ABB RAPID module: MonProgramme.mod

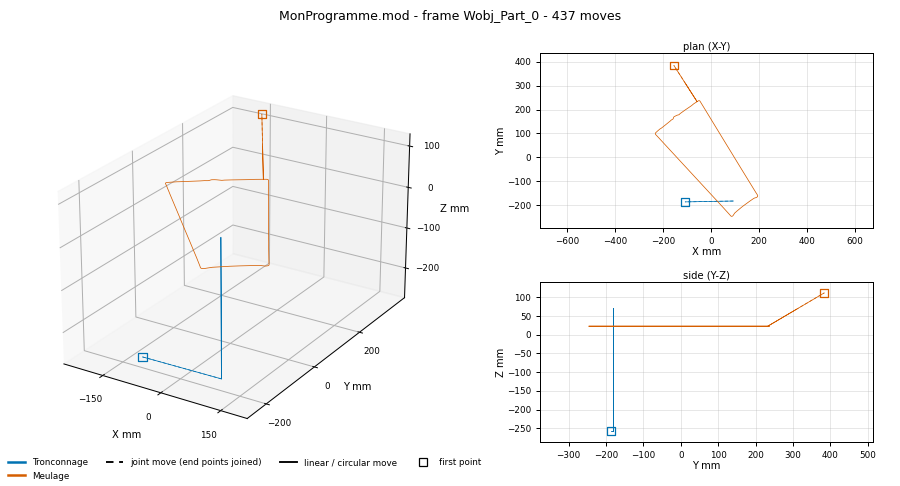
[picture p0: tool path of MonProgramme.mod in frame Wobj_Part_0, 437 of 442 moves have a stored position in this frame; points joined in program order, loops and branches not executed]
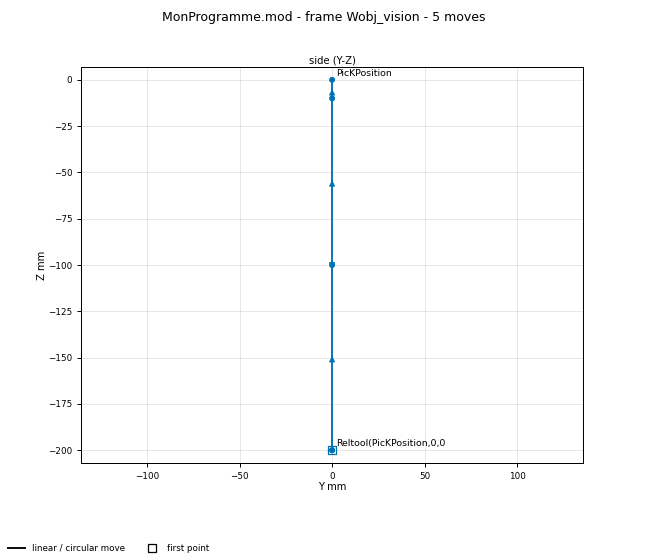
[picture p1: tool path of MonProgramme.mod in frame Wobj_vision, 5 of 442 moves have a stored position in this frame; points joined in program order, loops and branches not executed]
MODULE MonProgramme

    ! Nom         :MonProgramme
    ! Description :Pièce plate numero 1 famille 10
    ! Cree le     :30/03/2023 10:33:36

    CONST SPEEDDATA VitesseLente :=[10,500,0,0];
    CONST SPEEDDATA VitesseRapide :=[20,500,0,0];
    !
    !Point de prise
    PERS Robtarget PicKPosition := [[0,0,0],[0,0,0,0],[0,0,0,0],[9E9,9E9,9E9,9E9,9E9,9E9]];
    PERS Pose Ref := [[0,0,0],[1,0,0,0]];
    !
    !Declaration des points de meulage

    !Meulage_1 : Meulage du plan de joint
    CONST Robtarget Meulage_1_0 := [[-58.3575,232.789,23],[0.148181865705,-0.238974835253123,0.815584650429269,-0.505722098366382],[0,0,0,0],[8.999999E+09,8.999999E+09,8.999999E+09,8.999999E+09,8.999999E+09,8.999999E+09]];
    CONST Robtarget Meulage_1_1 := [[-61.8861,230.625,23],[0.148625433017615,-0.239693187884457,0.815376906988774,-0.505586941970947],[0,0,0,0],[8.999999E+09,8.999999E+09,8.999999E+09,8.999999E+09,8.999999E+09,8.999999E+09]];
    CONST Robtarget Meulage_1_2 := [[-62.4113,230.301,23],[0.149925832812002,-0.241798832684592,0.814763562882074,-0.505188980251654],[0,0,0,0],[8.999999E+09,8.999999E+09,8.999999E+09,8.999999E+09,8.999999E+09,8.999999E+09]];
    CONST Robtarget Meulage_1_3 := [[-62.698,230.118,23],[0.151989778330523,-0.245141375569821,0.81377802973829,-0.504549434230225],[0,0,0,0],[8.999999E+09,8.999999E+09,8.999999E+09,8.999999E+09,8.999999E+09,8.999999E+09]];
    CONST Robtarget Meulage_1_4 := [[-63.1019,229.854,23],[0.154659485743828,-0.249466287008623,0.812481437559476,-0.50370718551245],[0,0,0,0],[8.999999E+09,8.999999E+09,8.999999E+09,8.999999E+09,8.999999E+09,8.999999E+09]];
    CONST Robtarget Meulage_1_5 := [[-70.7437,224.925,23],[0.157674904224026,-0.254354542291001,0.810988113593647,-0.502733200618079],[0,0,0,0],[8.999999E+09,8.999999E+09,8.999999E+09,8.999999E+09,8.999999E+09,8.999999E+09]];
    CONST Robtarget Meulage_1_6 := [[-71.9304,224.189,23],[0.160716946471538,-0.259293185737598,0.80945258539058,-0.501720658286478],[0,0,0,0],[8.999999E+09,8.999999E+09,8.999999E+09,8.999999E+09,8.999999E+09,8.999999E+09]];
    CONST Robtarget Meulage_1_7 := [[-74.21,222.511,23],[0.163429453183647,-0.26370625584774,0.808060318676629,-0.500787725327893],[0,0,0,0],[8.999999E+09,8.999999E+09,8.999999E+09,8.999999E+09,8.999999E+09,8.999999E+09]];
    CONST Robtarget Meulage_1_8 := [[-74.4047,222.355,23],[0.165478565930098,-0.267054985800185,0.80699916691214,-0.50005082079734],[0,0,0,0],[8.999999E+09,8.999999E+09,8.999999E+09,8.999999E+09,8.999999E+09,8.999999E+09]];
    CONST Robtarget Meulage_1_9 := [[-75.4181,221.463,23],[0.166625756157986,-0.26895524483736,0.806413026211877,-0.499596802246629],[0,0,0,0],[8.999999E+09,8.999999E+09,8.999999E+09,8.999999E+09,8.999999E+09,8.999999E+09]];
    CONST Robtarget Meulage_1_10 := [[-77.7294,219.409,23],[0.16678460212446,-0.269265640729812,0.806359285274043,-0.49946332625017],[0,0,0,0],[8.999999E+09,8.999999E+09,8.999999E+09,8.999999E+09,8.999999E+09,8.999999E+09]];
    CONST Robtarget Meulage_1_11 := [[-79.8592,217.425,23],[0.166011121163228,-0.268074246853636,0.806809289446494,-0.499635143166319],[0,0,0,0],[8.999999E+09,8.999999E+09,8.999999E+09,8.999999E+09,8.999999E+09,8.999999E+09]];
    CONST Robtarget Meulage_1_12 := [[-80.9664,216.585,23],[0.164506342942007,-0.265705695049484,0.807649709633931,-0.500040091671002],[0,0,0,0],[8.999999E+09,8.999999E+09,8.999999E+09,8.999999E+09,8.999999E+09,8.999999E+09]];
    CONST Robtarget Meulage_1_13 := [[-81.6442,216.056,23],[0.162565848926237,-0.262638222690881,0.808715379393519,-0.500572615987993],[0,0,0,0],[8.999999E+09,8.999999E+09,8.999999E+09,8.999999E+09,8.999999E+09,8.999999E+09]];
    CONST Robtarget Meulage_1_14 := [[-83.4588,214.852,23],[0.160506269342085,-0.259380438725357,0.809832525449451,-0.501129530393781],[0,0,0,0],[8.999999E+09,8.999999E+09,8.999999E+09,8.999999E+09,8.999999E+09,8.999999E+09]];
    CONST Robtarget Meulage_1_15 := [[-85.6252,213.407,23],[0.158605509281455,-0.256380354449679,0.810856236167601,-0.501622936622658],[0,0,0,0],[8.999999E+09,8.999999E+09,8.999999E+09,8.999999E+09,8.999999E+09,8.999999E+09]];
    CONST Robtarget Meulage_1_16 := [[-88.6992,211.314,23],[0.157073467166774,-0.253977478744035,0.811683564072664,-0.501989201096328],[0,0,0,0],[8.999999E+09,8.999999E+09,8.999999E+09,8.999999E+09,8.999999E+09,8.999999E+09]];
    CONST Robtarget Meulage_1_17 := [[-97.9458,205.12,23],[0.156019831326172,-0.252351695101114,0.812266525129294,-0.502194709616629],[0,0,0,0],[8.999999E+09,8.999999E+09,8.999999E+09,8.999999E+09,8.999999E+09,8.999999E+09]];
    CONST Robtarget Meulage_1_18 := [[-98.0906,205.024,23],[0.155481024731552,-0.251559631951472,0.812589912996045,-0.502236035961128],[0,0,0,0],[8.999999E+09,8.999999E+09,8.999999E+09,8.999999E+09,8.999999E+09,8.999999E+09]];
    CONST Robtarget Meulage_1_19 := [[-98.2298,204.931,23],[0.15543444332337,-0.251566601297488,0.812668312025136,-0.502120098751883],[0,0,0,0],[8.999999E+09,8.999999E+09,8.999999E+09,8.999999E+09,8.999999E+09,8.999999E+09]];
    CONST Robtarget Meulage_1_20 := [[-106.087,199.59,23],[0.155835854786064,-0.252301771176396,0.812523766656786,-0.501860669152523],[0,0,0,0],[8.999999E+09,8.999999E+09,8.999999E+09,8.999999E+09,8.999999E+09,8.999999E+09]];
    CONST Robtarget Meulage_1_21 := [[-107.424,198.616,23],[0.156627171164782,-0.253671144300647,0.812182880878495,-0.501475670207466],[0,0,0,0],[8.999999E+09,8.999999E+09,8.999999E+09,8.999999E+09,8.999999E+09,8.999999E+09]];
    CONST Robtarget Meulage_1_22 := [[-108.97,197.494,23],[0.157776257270276,-0.255622208619674,0.811657634087461,-0.500974873750899],[0,0,0,0],[8.999999E+09,8.999999E+09,8.999999E+09,8.999999E+09,8.999999E+09,8.999999E+09]];
    CONST Robtarget Meulage_1_23 := [[-114.95,193.344,23],[0.159245499185872,-0.258095332379691,0.810963108965959,-0.500366372060639],[0,0,0,0],[8.999999E+09,8.999999E+09,8.999999E+09,8.999999E+09,8.999999E+09,8.999999E+09]];
    CONST Robtarget Meulage_1_24 := [[-116.539,192.217,23],[0.160993233363206,-0.261024743289672,0.810116382511968,-0.499658592428415],[0,0,0,0],[8.999999E+09,8.999999E+09,8.999999E+09,8.999999E+09,8.999999E+09,8.999999E+09]];
    CONST Robtarget Meulage_1_25 := [[-117.242,191.715,23],[0.162968822500786,-0.264326079213905,0.809136936165937,-0.498869026170308],[0,0,0,0],[8.999999E+09,8.999999E+09,8.999999E+09,8.999999E+09,8.999999E+09,8.999999E+09]];
    CONST Robtarget Meulage_1_26 := [[-122.753,187.734,23],[0.165068141160407,-0.26783129174422,0.808075887267558,-0.498028381072022],[0,0,0,0],[8.999999E+09,8.999999E+09,8.999999E+09,8.999999E+09,8.999999E+09,8.999999E+09]];
    CONST Robtarget Meulage_1_27 := [[-124.08,186.83,23],[0.167128719704548,-0.271277404998019,0.807019143914389,-0.497188758866435],[0,0,0,0],[8.999999E+09,8.999999E+09,8.999999E+09,8.999999E+09,8.999999E+09,8.999999E+09]];
    CONST Robtarget Meulage_1_28 := [[-124.769,186.441,23],[0.168925773409572,-0.274298901580079,0.806091509326518,-0.496427914466578],[0,0,0,0],[8.999999E+09,8.999999E+09,8.999999E+09,8.999999E+09,8.999999E+09,8.999999E+09]];
    CONST Robtarget Meulage_1_29 := [[-125.945,185.703,23],[0.170183715064392,-0.276447157139279,0.805451882761743,-0.495844468550427],[0,0,0,0],[8.999999E+09,8.999999E+09,8.999999E+09,8.999999E+09,8.999999E+09,8.999999E+09]];
    CONST Robtarget Meulage_1_30 := [[-127.541,184.735,23],[0.170563540523803,-0.277170778046338,0.805298374334778,-0.49555924644278],[0,0,0,0],[8.999999E+09,8.999999E+09,8.999999E+09,8.999999E+09,8.999999E+09,8.999999E+09]];
    CONST Robtarget Meulage_1_31 := [[-128.688,183.725,23],[0.169740584331575,-0.275939588736474,0.805816183323026,-0.495687155465454],[0,0,0,0],[8.999999E+09,8.999999E+09,8.999999E+09,8.999999E+09,8.999999E+09,8.999999E+09]];
    CONST Robtarget Meulage_1_32 := [[-129.358,183.125,23],[0.167388097421785,-0.272218246565665,0.807174270619609,-0.496334713603564],[0,0,0,0],[8.999999E+09,8.999999E+09,8.999999E+09,8.999999E+09,8.999999E+09,8.999999E+09]];
    CONST Robtarget Meulage_1_33 := [[-129.919,182.398,23],[0.163240285146969,-0.265572531090826,0.809477525318781,-0.497564042148276],[0,0,0,0],[8.999999E+09,8.999999E+09,8.999999E+09,8.999999E+09,8.999999E+09,8.999999E+09]];
    CONST Robtarget Meulage_1_34 := [[-131.979,179.902,23],[0.157173550553764,-0.255799420019378,0.812711409516704,-0.499362890657131],[0,0,0,0],[8.999999E+09,8.999999E+09,8.999999E+09,8.999999E+09,8.999999E+09,8.999999E+09]];
    CONST Robtarget Meulage_1_35 := [[-134.06,178.158,23],[0.149236843350465,-0.242970650244417,0.816726929966982,-0.501648033558692],[0,0,0,0],[8.999999E+09,8.999999E+09,8.999999E+09,8.999999E+09,8.999999E+09,8.999999E+09]];
    CONST Robtarget Meulage_1_36 := [[-134.165,178.081,23],[0.139752269082147,-0.227609102553757,0.821225804183011,-0.504233654435155],[0,0,0,0],[8.999999E+09,8.999999E+09,8.999999E+09,8.999999E+09,8.999999E+09,8.999999E+09]];
    CONST Robtarget Meulage_1_37 := [[-134.441,178.011,23],[0.129325108544261,-0.210699865727179,0.825809425898454,-0.50687214855408],[0,0,0,0],[8.999999E+09,8.999999E+09,8.999999E+09,8.999999E+09,8.999999E+09,8.999999E+09]];
    CONST Robtarget Meulage_1_38 := [[-136.03,177.529,23],[0.118837759157301,-0.19367817259203,0.830046350348129,-0.509302865428455],[0,0,0,0],[8.999999E+09,8.999999E+09,8.999999E+09,8.999999E+09,8.999999E+09,8.999999E+09]];
    CONST Robtarget Meulage_1_39 := [[-137.058,177.428,23],[0.109319526610547,-0.17822251532365,0.833577665229546,-0.511306417096261],[0,0,0,0],[8.999999E+09,8.999999E+09,8.999999E+09,8.999999E+09,8.999999E+09,8.999999E+09]];
    CONST Robtarget Meulage_1_40 := [[-137.767,177.244,23],[0.101834444100147,-0.166069093537888,0.836154474307736,-0.512734333999072],[0,0,0,0],[8.999999E+09,8.999999E+09,8.999999E+09,8.999999E+09,8.999999E+09,8.999999E+09]];
    CONST Robtarget Meulage_1_41 := [[-138.926,177.032,23],[0.0972609331651995,-0.158655399925333,0.837659570016408,-0.513512628583069],[0,0,0,0],[8.999999E+09,8.999999E+09,8.999999E+09,8.999999E+09,8.999999E+09,8.999999E+09]];
    CONST Robtarget Meulage_1_42 := [[-141.055,176.503,23],[0.0962333946459954,-0.157018976046454,0.838027811217633,-0.513608374680567],[0,0,0,0],[8.999999E+09,8.999999E+09,8.999999E+09,8.999999E+09,8.999999E+09,8.999999E+09]];
    CONST Robtarget Meulage_1_43 := [[-142.608,175.886,23],[0.0991568880059853,-0.161825994734284,0.837166926328479,-0.512963737949337],[0,0,0,0],[8.999999E+09,8.999999E+09,8.999999E+09,8.999999E+09,8.999999E+09,8.999999E+09]];
    CONST Robtarget Meulage_1_44 := [[-143.78,175.336,23],[0.106181630726738,-0.173325871848446,0.834910311212505,-0.511476661906704],[0,0,0,0],[8.999999E+09,8.999999E+09,8.999999E+09,8.999999E+09,8.999999E+09,8.999999E+09]];
    CONST Robtarget Meulage_1_45 := [[-145.369,174.717,23],[0.117249638213944,-0.191423627162767,0.830986199154812,-0.50899062281813],[0,0,0,0],[8.999999E+09,8.999999E+09,8.999999E+09,8.999999E+09,8.999999E+09,8.999999E+09]];
    CONST Robtarget Meulage_1_46 := [[-147.738,173.712,23],[0.132042011999882,-0.215600202183316,0.825073354624242,-0.50530725244611],[0,0,0,0],[8.999999E+09,8.999999E+09,8.999999E+09,8.999999E+09,8.999999E+09,8.999999E+09]];
    CONST Robtarget Meulage_1_47 := [[-149.854,172.757,23],[0.149936736958957,-0.24483795390417,0.816893265959095,-0.500258676355347],[0,0,0,0],[8.999999E+09,8.999999E+09,8.999999E+09,8.999999E+09,8.999999E+09,8.999999E+09]];
    CONST Robtarget Meulage_1_48 := [[-154.216,170.145,23],[0.169830628833517,-0.277333648028576,0.806449481811435,-0.493844953874434],[0,0,0,0],[8.999999E+09,8.999999E+09,8.999999E+09,8.999999E+09,8.999999E+09,8.999999E+09]];
    CONST Robtarget Meulage_1_49 := [[-154.437,169.987,23],[0.190173723560722,-0.31054786386223,0.794246164394551,-0.48638154720569],[0,0,0,0],[8.999999E+09,8.999999E+09,8.999999E+09,8.999999E+09,8.999999E+09,8.999999E+09]];
    CONST Robtarget Meulage_1_50 := [[-154.594,169.835,23],[0.20901486158858,-0.341289935912337,0.781510811666196,-0.478617612012871],[0,0,0,0],[8.999999E+09,8.999999E+09,8.999999E+09,8.999999E+09,8.999999E+09,8.999999E+09]];
    CONST Robtarget Meulage_1_51 := [[-155.629,168.85,23],[0.224377432981166,-0.366324782084454,0.770058471733467,-0.471668179667737],[0,0,0,0],[8.999999E+09,8.999999E+09,8.999999E+09,8.999999E+09,8.999999E+09,8.999999E+09]];
    CONST Robtarget Meulage_1_52 := [[-156.133,167.795,23],[0.234664546304594,-0.383040973631614,0.761827965710797,-0.466722951961817],[0,0,0,0],[8.999999E+09,8.999999E+09,8.999999E+09,8.999999E+09,8.999999E+09,8.999999E+09]];
    CONST Robtarget Meulage_1_53 := [[-156.63,166.376,23],[0.238858700263915,-0.389779733116246,0.758330223876227,-0.464708029321522],[0,0,0,0],[8.999999E+09,8.999999E+09,8.999999E+09,8.999999E+09,8.999999E+09,8.999999E+09]];
    CONST Robtarget Meulage_1_54 := [[-157.04,165.499,23],[0.236694401045912,-0.386113732187725,0.760112613369517,-0.465962188730101],[0,0,0,0],[8.999999E+09,8.999999E+09,8.999999E+09,8.999999E+09,8.999999E+09,8.999999E+09]];
    CONST Robtarget Meulage_1_55 := [[-157.361,164.48,23],[0.228724405566161,-0.372950235137066,0.766544447802728,-0.470109431890516],[0,0,0,0],[8.999999E+09,8.999999E+09,8.999999E+09,8.999999E+09,8.999999E+09,8.999999E+09]];
    CONST Robtarget Meulage_1_56 := [[-157.884,162.467,23],[0.216369665365497,-0.352618880208087,0.775971980241673,-0.476142393733466],[0,0,0,0],[8.999999E+09,8.999999E+09,8.999999E+09,8.999999E+09,8.999999E+09,8.999999E+09]];
    CONST Robtarget Meulage_1_57 := [[-158.273,161.139,23],[0.201902642085932,-0.328839509863673,0.786188645105272,-0.482708311694418],[0,0,0,0],[8.999999E+09,8.999999E+09,8.999999E+09,8.999999E+09,8.999999E+09,8.999999E+09]];
    CONST Robtarget Meulage_1_58 := [[-159.533,159.945,23],[0.187867683973008,-0.305761928032033,0.795269209582019,-0.488633053502874],[0,0,0,0],[8.999999E+09,8.999999E+09,8.999999E+09,8.999999E+09,8.999999E+09,8.999999E+09]];
    CONST Robtarget Meulage_1_59 := [[-160.756,159.116,23],[0.176380566922609,-0.286828351785849,0.802086672165354,-0.493230536928301],[0,0,0,0],[8.999999E+09,8.999999E+09,8.999999E+09,8.999999E+09,8.999999E+09,8.999999E+09]];
    CONST Robtarget Meulage_1_60 := [[-164.86,156.999,23],[0.168574311156337,-0.273876845029363,0.806369203223988,-0.496329410237636],[0,0,0,0],[8.999999E+09,8.999999E+09,8.999999E+09,8.999999E+09,8.999999E+09,8.999999E+09]];
    CONST Robtarget Meulage_1_61 := [[-164.955,156.947,23],[0.164588289155838,-0.267117123661376,0.80837176084268,-0.498090587736541],[0,0,0,0],[8.999999E+09,8.999999E+09,8.999999E+09,8.999999E+09,8.999999E+09,8.999999E+09]];
    CONST Robtarget Meulage_1_62 := [[-164.971,156.936,23],[0.163859430505866,-0.265620070980564,0.80857322311266,-0.498803977321532],[0,0,0,0],[8.999999E+09,8.999999E+09,8.999999E+09,8.999999E+09,8.999999E+09,8.999999E+09]];
    CONST Robtarget Meulage_1_63 := [[-166.361,155.833,23],[0.165381377584628,-0.267732246634111,0.807548604928368,-0.498832331288489],[0,0,0,0],[8.999999E+09,8.999999E+09,8.999999E+09,8.999999E+09,8.999999E+09,8.999999E+09]];
    CONST Robtarget Meulage_1_64 := [[-168.503,153.688,23],[0.168104311079277,-0.271741892549473,0.805844559691503,-0.498509608779811],[0,0,0,0],[8.999999E+09,8.999999E+09,8.999999E+09,8.999999E+09,8.999999E+09,8.999999E+09]];
    CONST Robtarget Meulage_1_65 := [[-168.732,153.484,23],[0.171095363611995,-0.276129456875717,0.803948321874422,-0.498142545213015],[0,0,0,0],[8.999999E+09,8.999999E+09,8.999999E+09,8.999999E+09,8.999999E+09,8.999999E+09]];
    CONST Robtarget Meulage_1_66 := [[-168.989,153.24,23],[0.173727216355865,-0.279874854590491,0.802203981283839,-0.497953504333037],[0,0,0,0],[8.999999E+09,8.999999E+09,8.999999E+09,8.999999E+09,8.999999E+09,8.999999E+09]];
    CONST Robtarget Meulage_1_67 := [[-170.912,151.541,23],[0.175699268719496,-0.282498394157683,0.800792871461658,-0.498051404260601],[0,0,0,0],[8.999999E+09,8.999999E+09,8.999999E+09,8.999999E+09,8.999999E+09,8.999999E+09]];
    CONST Robtarget Meulage_1_68 := [[-173.64,149.409,23],[0.176961646667263,-0.28391777107171,0.799750367106998,-0.498472291296824],[0,0,0,0],[8.999999E+09,8.999999E+09,8.999999E+09,8.999999E+09,8.999999E+09,8.999999E+09]];
    CONST Robtarget Meulage_1_69 := [[-178.74,145.33,23],[0.177643876260341,-0.284343906869504,0.799006395151077,-0.499179302817204],[0,0,0,0],[8.999999E+09,8.999999E+09,8.999999E+09,8.999999E+09,8.999999E+09,8.999999E+09]];
    CONST Robtarget Meulage_1_70 := [[-181.409,143.189,23],[0.177885375662456,-0.284001180466343,0.798479267411956,-0.50013096498059],[0,0,0,0],[8.999999E+09,8.999999E+09,8.999999E+09,8.999999E+09,8.999999E+09,8.999999E+09]];
    CONST Robtarget Meulage_1_71 := [[-182.06,142.684,23],[0.177829054554651,-0.283120776982402,0.798084298268948,-0.501279269323638],[0,0,0,0],[8.999999E+09,8.999999E+09,8.999999E+09,8.999999E+09,8.999999E+09,8.999999E+09]];
    CONST Robtarget Meulage_1_72 := [[-184.754,140.501,23],[0.177508601805971,-0.281756942245647,0.797796917662663,-0.502616951513999],[0,0,0,0],[8.999999E+09,8.999999E+09,8.999999E+09,8.999999E+09,8.999999E+09,8.999999E+09]];
    CONST Robtarget Meulage_1_73 := [[-185.572,139.809,23],[0.176889769752061,-0.279853929726552,0.797628079870075,-0.504163895550293],[0,0,0,0],[8.999999E+09,8.999999E+09,8.999999E+09,8.999999E+09,8.999999E+09,8.999999E+09]];
    CONST Robtarget Meulage_1_74 := [[-190.016,136.046,23],[0.175866828136052,-0.277249856410041,0.797628532251201,-0.505956619109554],[0,0,0,0],[8.999999E+09,8.999999E+09,8.999999E+09,8.999999E+09,8.999999E+09,8.999999E+09]];
    CONST Robtarget Meulage_1_75 := [[-194.685,132.291,23],[0.174337183351613,-0.273784872962367,0.797838615743534,-0.508037334323422],[0,0,0,0],[8.999999E+09,8.999999E+09,8.999999E+09,8.999999E+09,8.999999E+09,8.999999E+09]];
    CONST Robtarget Meulage_1_76 := [[-195.72,131.454,23],[0.172252983388396,-0.269393907820685,0.798265969451153,-0.51041872434219],[0,0,0,0],[8.999999E+09,8.999999E+09,8.999999E+09,8.999999E+09,8.999999E+09,8.999999E+09]];
    CONST Robtarget Meulage_1_77 := [[-198.083,129.418,23],[0.169683326213003,-0.264196789696462,0.798852292573998,-0.513071768633436],[0,0,0,0],[8.999999E+09,8.999999E+09,8.999999E+09,8.999999E+09,8.999999E+09,8.999999E+09]];
    CONST Robtarget Meulage_1_78 := [[-202.369,125.72,23],[0.166815627644645,-0.258495591847161,0.799480014112797,-0.515930501524489],[0,0,0,0],[8.999999E+09,8.999999E+09,8.999999E+09,8.999999E+09,8.999999E+09,8.999999E+09]];
    CONST Robtarget Meulage_1_79 := [[-204.09,124.347,23],[0.163975032533586,-0.252798071370166,0.799971563273555,-0.518893844414056],[0,0,0,0],[8.999999E+09,8.999999E+09,8.999999E+09,8.999999E+09,8.999999E+09,8.999999E+09]];
    CONST Robtarget Meulage_1_80 := [[-205.316,123.493,23],[0.161593456334009,-0.247768082539381,0.800117515820452,-0.521833779111794],[0,0,0,0],[8.999999E+09,8.999999E+09,8.999999E+09,8.999999E+09,8.999999E+09,8.999999E+09]];
    CONST Robtarget Meulage_1_81 := [[-206.826,122.557,23],[0.160103775598754,-0.24405859141989,0.799730148614511,-0.524627367176147],[0,0,0,0],[8.999999E+09,8.999999E+09,8.999999E+09,8.999999E+09,8.999999E+09,8.999999E+09]];
    CONST Robtarget Meulage_1_82 := [[-207.594,122.163,23],[0.159904315850039,-0.242251029651226,0.7986476248747,-0.52716887207749],[0,0,0,0],[8.999999E+09,8.999999E+09,8.999999E+09,8.999999E+09,8.999999E+09,8.999999E+09]];
    CONST Robtarget Meulage_1_83 := [[-211.136,120.249,23],[0.161232247651532,-0.24266569861192,0.796778854775407,-0.529396805446742],[0,0,0,0],[8.999999E+09,8.999999E+09,8.999999E+09,8.999999E+09,8.999999E+09,8.999999E+09]];
    CONST Robtarget Meulage_1_84 := [[-211.486,120.042,23],[0.164173102785519,-0.24538461188339,0.794087822782301,-0.531279694964412],[0,0,0,0],[8.999999E+09,8.999999E+09,8.999999E+09,8.999999E+09,8.999999E+09,8.999999E+09]];
    CONST Robtarget Meulage_1_85 := [[-212.259,119.628,23],[0.168636469158135,-0.25021946193254,0.790598991725033,-0.532827548483962],[0,0,0,0],[8.999999E+09,8.999999E+09,8.999999E+09,8.999999E+09,8.999999E+09,8.999999E+09]];
    CONST Robtarget Meulage_1_86 := [[-213.995,118.332,23],[0.17444356931549,-0.256852295719363,0.786364538293094,-0.534066617776522],[0,0,0,0],[8.999999E+09,8.999999E+09,8.999999E+09,8.999999E+09,8.999999E+09,8.999999E+09]];
    CONST Robtarget Meulage_1_87 := [[-215.118,117.432,23],[0.181390149627336,-0.264937976302254,0.781447432216692,-0.535019058551167],[0,0,0,0],[8.999999E+09,8.999999E+09,8.999999E+09,8.999999E+09,8.999999E+09,8.999999E+09]];
    CONST Robtarget Meulage_1_88 := [[-219.68,113.42,23],[0.189445681651388,-0.274384787928736,0.775819880233113,-0.535655519239765],[0,0,0,0],[8.999999E+09,8.999999E+09,8.999999E+09,8.999999E+09,8.999999E+09,8.999999E+09]];
    CONST Robtarget Meulage_1_89 := [[-220.066,113.076,23],[0.198828497289454,-0.285462403668641,0.769319367664705,-0.535841539350318],[0,0,0,0],[8.999999E+09,8.999999E+09,8.999999E+09,8.999999E+09,8.999999E+09,8.999999E+09]];
    CONST Robtarget Meulage_1_90 := [[-222.535,110.973,23],[0.210159368146795,-0.29899638785888,0.761528392678817,-0.535265081218176],[0,0,0,0],[8.999999E+09,8.999999E+09,8.999999E+09,8.999999E+09,8.999999E+09,8.999999E+09]];
    CONST Robtarget Meulage_1_91 := [[-223.217,110.388,23],[0.224421010770944,-0.316294163357458,0.751731894064707,-0.53337826314581],[0,0,0,0],[8.999999E+09,8.999999E+09,8.999999E+09,8.999999E+09,8.999999E+09,8.999999E+09]];
    CONST Robtarget Meulage_1_92 := [[-223.432,110.2,23],[0.2428257751573,-0.338928357428283,0.738873325024166,-0.529367000310706],[0,0,0,0],[8.999999E+09,8.999999E+09,8.999999E+09,8.999999E+09,8.999999E+09,8.999999E+09]];
    CONST Robtarget Meulage_1_93 := [[-224.086,109.631,23],[0.266639538914918,-0.368473967425196,0.721490518015019,-0.522093597003062],[0,0,0,0],[8.999999E+09,8.999999E+09,8.999999E+09,8.999999E+09,8.999999E+09,8.999999E+09]];
    CONST Robtarget Meulage_1_94 := [[-228.959,105.341,23],[0.296633408139784,-0.405758573815811,0.697897215860017,-0.51020395632058],[0,0,0,0],[8.999999E+09,8.999999E+09,8.999999E+09,8.999999E+09,8.999999E+09,8.999999E+09]];
    CONST Robtarget Meulage_1_95 := [[-230.28,104.199,23],[0.332446608572302,-0.450035148768836,0.666652847465604,-0.492464819339807],[0,0,0,0],[8.999999E+09,8.999999E+09,8.999999E+09,8.999999E+09,8.999999E+09,8.999999E+09]];
    CONST Robtarget Meulage_1_96 := [[-231.158,103.201,23],[0.372007037225721,-0.498286041084704,0.62754961066334,-0.468511762574819],[0,0,0,0],[8.999999E+09,8.999999E+09,8.999999E+09,8.999999E+09,8.999999E+09,8.999999E+09]];
    CONST Robtarget Meulage_1_97 := [[-232.151,102.067,23],[0.411728777245195,-0.5456127649428,0.582643773137358,-0.43967301298114],[0,0,0,0],[8.999999E+09,8.999999E+09,8.999999E+09,8.999999E+09,8.999999E+09,8.999999E+09]];
    CONST Robtarget Meulage_1_98 := [[-232.796,99.9633,23],[0.447997467343063,-0.587290838043957,0.535950238760348,-0.408833807771023],[0,0,0,0],[8.999999E+09,8.999999E+09,8.999999E+09,8.999999E+09,8.999999E+09,8.999999E+09]];
    CONST Robtarget Meulage_1_99 := [[-232.94,99.3444,23],[0.478708689081828,-0.620768093986057,0.491662236257723,-0.379148005302059],[0,0,0,0],[8.999999E+09,8.999999E+09,8.999999E+09,8.999999E+09,8.999999E+09,8.999999E+09]];
    CONST Robtarget Meulage_1_100 := [[-232.9,98.7836,23],[0.503565532327161,-0.645935886127157,0.452492698047789,-0.352759045069889],[0,0,0,0],[8.999999E+09,8.999999E+09,8.999999E+09,8.999999E+09,8.999999E+09,8.999999E+09]];
    CONST Robtarget Meulage_1_101 := [[-232.43,97.6663,23],[0.523316087361497,-0.664031317820012,0.419443923999624,-0.330559338519833],[0,0,0,0],[8.999999E+09,8.999999E+09,8.999999E+09,8.999999E+09,8.999999E+09,8.999999E+09]];
    CONST Robtarget Meulage_1_102 := [[-231.726,95.9117,23],[0.539002339752526,-0.676610402546008,0.392385905017713,-0.31258301689513],[0,0,0,0],[8.999999E+09,8.999999E+09,8.999999E+09,8.999999E+09,8.999999E+09,8.999999E+09]];
    CONST Robtarget Meulage_1_103 := [[-231.567,95.7075,23],[0.551578119930835,-0.685059014028228,0.370661133221146,-0.298439356036454],[0,0,0,0],[8.999999E+09,8.999999E+09,8.999999E+09,8.999999E+09,8.999999E+09,8.999999E+09]];
    CONST Robtarget Meulage_1_104 := [[-229.121,92.9592,23],[0.561769116597744,-0.690428997992429,0.353527443928271,-0.287648404754317],[0,0,0,0],[8.999999E+09,8.999999E+09,8.999999E+09,8.999999E+09,8.999999E+09,8.999999E+09]];
    CONST Robtarget Meulage_1_105 := [[-227.691,91.6359,23],[0.570128958343692,-0.69352255369769,0.340224337828433,-0.279690611783406],[0,0,0,0],[8.999999E+09,8.999999E+09,8.999999E+09,8.999999E+09,8.999999E+09,8.999999E+09]];
    CONST Robtarget Meulage_1_106 := [[-223.426,87.372,23],[0.577070461009341,-0.694933127142454,0.330057942011735,-0.274079161457881],[0,0,0,0],[8.999999E+09,8.999999E+09,8.999999E+09,8.999999E+09,8.999999E+09,8.999999E+09]];
    CONST Robtarget Meulage_1_107 := [[-223.34,87.278,23],[0.582894421628478,-0.6950996893225,0.322432572506357,-0.270384450967689],[0,0,0,0],[8.999999E+09,8.999999E+09,8.999999E+09,8.999999E+09,8.999999E+09,8.999999E+09]];
    CONST Robtarget Meulage_1_108 := [[-223.088,87.002,23],[0.587858784719537,-0.694391357404035,0.316754794514291,-0.268158707005497],[0,0,0,0],[8.999999E+09,8.999999E+09,8.999999E+09,8.999999E+09,8.999999E+09,8.999999E+09]];
    CONST Robtarget Meulage_1_109 := [[-222.82,86.7227,23],[0.592161137568373,-0.693084135536069,0.312533953200178,-0.267024523815734],[0,0,0,0],[8.999999E+09,8.999999E+09,8.999999E+09,8.999999E+09,8.999999E+09,8.999999E+09]];
    CONST Robtarget Meulage_1_110 := [[-221.051,84.8092,23],[0.595963533668866,-0.691407608350969,0.309336353326606,-0.266634592958058],[0,0,0,0],[8.999999E+09,8.999999E+09,8.999999E+09,8.999999E+09,8.999999E+09,8.999999E+09]];
    CONST Robtarget Meulage_1_111 := [[-219.779,83.3882,23],[0.59938716449273,-0.689529144008234,0.306831249380014,-0.26671927378526],[0,0,0,0],[8.999999E+09,8.999999E+09,8.999999E+09,8.999999E+09,8.999999E+09,8.999999E+09]];
    CONST Robtarget Meulage_1_112 := [[-215.703,78.7371,23],[0.602509293513914,-0.687562677408874,0.3047973274786,-0.267093064353249],[0,0,0,0],[8.999999E+09,8.999999E+09,8.999999E+09,8.999999E+09,8.999999E+09,8.999999E+09]];
    CONST Robtarget Meulage_1_113 := [[-211.258,73.9555,23],[0.605382483164007,-0.685574643056103,0.303095711327686,-0.26764238762095],[0,0,0,0],[8.999999E+09,8.999999E+09,8.999999E+09,8.999999E+09,8.999999E+09,8.999999E+09]];
    CONST Robtarget Meulage_1_114 := [[-210.307,72.9122,23],[0.608038027534512,-0.683615226022337,0.301633168960238,-0.268286062264468],[0,0,0,0],[8.999999E+09,8.999999E+09,8.999999E+09,8.999999E+09,8.999999E+09,8.999999E+09]];
    CONST Robtarget Meulage_1_115 := [[-209.267,71.7626,23],[0.610492412702795,-0.681712367617464,0.300360453260437,-0.268981151731671],[0,0,0,0],[8.999999E+09,8.999999E+09,8.999999E+09,8.999999E+09,8.999999E+09,8.999999E+09]];
    CONST Robtarget Meulage_1_116 := [[-207.4,69.8087,23],[0.612756417865593,-0.679877891800581,0.299253289474695,-0.269709275598558],[0,0,0,0],[8.999999E+09,8.999999E+09,8.999999E+09,8.999999E+09,8.999999E+09,8.999999E+09]];
    CONST Robtarget Meulage_1_117 := [[-206.832,69.1988,23],[0.614837190252696,-0.678123547872162,0.298292338651236,-0.270453996098077],[0,0,0,0],[8.999999E+09,8.999999E+09,8.999999E+09,8.999999E+09,8.999999E+09,8.999999E+09]];
    CONST Robtarget Meulage_1_118 := [[-200.176,61.9772,23],[0.616740909593886,-0.676449934483326,0.297471214007645,-0.271213962412757],[0,0,0,0],[8.999999E+09,8.999999E+09,8.999999E+09,8.999999E+09,8.999999E+09,8.999999E+09]];
    CONST Robtarget Meulage_1_119 := [[-199.934,61.7141,23],[0.618478833410479,-0.674866517772944,0.296767228716791,-0.271971189231489],[0,0,0,0],[8.999999E+09,8.999999E+09,8.999999E+09,8.999999E+09,8.999999E+09,8.999999E+09]];
    CONST Robtarget Meulage_1_120 := [[-197.792,59.3246,23],[0.620059903950667,-0.67338053016784,0.296163128757491,-0.272711896088423],[0,0,0,0],[8.999999E+09,8.999999E+09,8.999999E+09,8.999999E+09,8.999999E+09,8.999999E+09]];
    CONST Robtarget Meulage_1_121 := [[-195.233,56.5182,23],[0.621501349254072,-0.671998364474201,0.295631278847074,-0.273416199202993],[0,0,0,0],[8.999999E+09,8.999999E+09,8.999999E+09,8.999999E+09,8.999999E+09,8.999999E+09]];
    CONST Robtarget Meulage_1_122 := [[-188.599,49.2598,23],[0.622819292554205,-0.670729522959678,0.295142321353333,-0.274060296283006],[0,0,0,0],[8.999999E+09,8.999999E+09,8.999999E+09,8.999999E+09,8.999999E+09,8.999999E+09]];
    CONST Robtarget Meulage_1_123 := [[-187.651,48.2771,23],[0.624035696410943,-0.669584173737313,0.294658328691099,-0.274614189761559],[0,0,0,0],[8.999999E+09,8.999999E+09,8.999999E+09,8.999999E+09,8.999999E+09,8.999999E+09]];
    CONST Robtarget Meulage_1_124 := [[-182.824,43.076,23],[0.625171095465849,-0.668570442383503,0.294145313074155,-0.275051267515101],[0,0,0,0],[8.999999E+09,8.999999E+09,8.999999E+09,8.999999E+09,8.999999E+09,8.999999E+09]];
    CONST Robtarget Meulage_1_125 := [[-181.69,41.843,23],[0.62624331181891,-0.667697199381823,0.293572029798568,-0.275345651245306],[0,0,0,0],[8.999999E+09,8.999999E+09,8.999999E+09,8.999999E+09,8.999999E+09,8.999999E+09]];
    CONST Robtarget Meulage_1_126 := [[-181.443,41.5678,23],[0.627265450659906,-0.666961618720308,0.292925058677238,-0.275490768559218],[0,0,0,0],[8.999999E+09,8.999999E+09,8.999999E+09,8.999999E+09,8.999999E+09,8.999999E+09]];
    CONST Robtarget Meulage_1_127 := [[-176.385,36.0713,23],[0.628242318577727,-0.666355686476183,0.292206973476687,-0.275493689402372],[0,0,0,0],[8.999999E+09,8.999999E+09,8.999999E+09,8.999999E+09,8.999999E+09,8.999999E+09]];
    CONST Robtarget Meulage_1_128 := [[-171.125,30.3489,23],[0.629173189579371,-0.665862579201927,0.291436265907064,-0.2753779694297],[0,0,0,0],[8.999999E+09,8.999999E+09,8.999999E+09,8.999999E+09,8.999999E+09,8.999999E+09]];
    CONST Robtarget Meulage_1_129 := [[-169.998,29.1159,23],[0.630050361006692,-0.665459118406619,0.290646995480448,-0.275181809615046],[0,0,0,0],[8.999999E+09,8.999999E+09,8.999999E+09,8.999999E+09,8.999999E+09,8.999999E+09]];
    CONST Robtarget Meulage_1_130 := [[-168.096,27.0444,23],[0.630863332605395,-0.665122211334356,0.289876869623482,-0.274945994735334],[0,0,0,0],[8.999999E+09,8.999999E+09,8.999999E+09,8.999999E+09,8.999999E+09,8.999999E+09]];
    CONST Robtarget Meulage_1_131 := [[-162.394,20.9104,23],[0.631604399753361,-0.664825496754764,0.289163112744995,-0.274713733374587],[0,0,0,0],[8.999999E+09,8.999999E+09,8.999999E+09,8.999999E+09,8.999999E+09,8.999999E+09]];
    CONST Robtarget Meulage_1_132 := [[-161.776,20.2388,23],[0.632263342849469,-0.664552175173201,0.288536887309725,-0.27451764319074],[0,0,0,0],[8.999999E+09,8.999999E+09,8.999999E+09,8.999999E+09,8.999999E+09,8.999999E+09]];
    CONST Robtarget Meulage_1_133 := [[-158.854,17.0923,23],[0.632843875046805,-0.664284119518685,0.288011681350255,-0.274380228472878],[0,0,0,0],[8.999999E+09,8.999999E+09,8.999999E+09,8.999999E+09,8.999999E+09,8.999999E+09]];
    CONST Robtarget Meulage_1_134 := [[-154.596,12.5439,23],[0.633346575777437,-0.664017003833627,0.287591366797009,-0.274307745633689],[0,0,0,0],[8.999999E+09,8.999999E+09,8.999999E+09,8.999999E+09,8.999999E+09,8.999999E+09]];
    CONST Robtarget Meulage_1_135 := [[-153.776,11.6279,23],[0.633781115990899,-0.663746048519823,0.28726773206263,-0.274298979588412],[0,0,0,0],[8.999999E+09,8.999999E+09,8.999999E+09,8.999999E+09,8.999999E+09,8.999999E+09]];
    CONST Robtarget Meulage_1_136 := [[-153.473,11.3104,23],[0.63415568454973,-0.663472030896534,0.287028921126526,-0.274346187158186],[0,0,0,0],[8.999999E+09,8.999999E+09,8.999999E+09,8.999999E+09,8.999999E+09,8.999999E+09]];
    CONST Robtarget Meulage_1_137 := [[-145.759,2.88919,23],[0.634481353232698,-0.663197107524958,0.286857673845988,-0.274437030894525],[0,0,0,0],[8.999999E+09,8.999999E+09,8.999999E+09,8.999999E+09,8.999999E+09,8.999999E+09]];
    CONST Robtarget Meulage_1_138 := [[-142.77,-0.315796,23],[0.634770280934764,-0.662919757939801,0.286738871676358,-0.274563115594222],[0,0,0,0],[8.999999E+09,8.999999E+09,8.999999E+09,8.999999E+09,8.999999E+09,8.999999E+09]];
    CONST Robtarget Meulage_1_139 := [[-138.619,-4.8035,23],[0.635023875559061,-0.662641312902346,0.286669253829191,-0.274721507738327],[0,0,0,0],[8.999999E+09,8.999999E+09,8.999999E+09,8.999999E+09,8.999999E+09,8.999999E+09]];
    CONST Robtarget Meulage_1_140 := [[-134.066,-9.70471,23],[0.635248005690691,-0.66235609548842,0.286646416344673,-0.274914906893191],[0,0,0,0],[8.999999E+09,8.999999E+09,8.999999E+09,8.999999E+09,8.999999E+09,8.999999E+09]];
    CONST Robtarget Meulage_1_141 := [[-128.009,-16.0721,23],[0.635439108402307,-0.662057725457776,0.286681529130601,-0.275155244416489],[0,0,0,0],[8.999999E+09,8.999999E+09,8.999999E+09,8.999999E+09,8.999999E+09,8.999999E+09]];
    CONST Robtarget Meulage_1_142 := [[-127.888,-16.2024,23],[0.635595973119153,-0.661739307296436,0.286782971357072,-0.27545303678333],[0,0,0,0],[8.999999E+09,8.999999E+09,8.999999E+09,8.999999E+09,8.999999E+09,8.999999E+09]];
    CONST Robtarget Meulage_1_143 := [[-127.769,-16.3286,23],[0.635720378305369,-0.661394553498304,0.286954326659855,-0.275815263575546],[0,0,0,0],[8.999999E+09,8.999999E+09,8.999999E+09,8.999999E+09,8.999999E+09,8.999999E+09]];
    CONST Robtarget Meulage_1_144 := [[-127.247,-16.8825,23],[0.635813299906298,-0.66102553152337,0.287191922667538,-0.276238110859151],[0,0,0,0],[8.999999E+09,8.999999E+09,8.999999E+09,8.999999E+09,8.999999E+09,8.999999E+09]];
    CONST Robtarget Meulage_1_145 := [[-122.136,-22.3277,23],[0.635885033980666,-0.660638637348887,0.287475080609727,-0.276703618389144],[0,0,0,0],[8.999999E+09,8.999999E+09,8.999999E+09,8.999999E+09,8.999999E+09,8.999999E+09]];
    CONST Robtarget Meulage_1_146 := [[-121.816,-22.6767,23],[0.635949263411385,-0.660244685414154,0.287774278125211,-0.277184874404061],[0,0,0,0],[8.999999E+09,8.999999E+09,8.999999E+09,8.999999E+09,8.999999E+09,8.999999E+09]];
    CONST Robtarget Meulage_1_147 := [[-115.802,-29.1783,23],[0.636024855969158,-0.659860035049179,0.288047720697922,-0.277642985387781],[0,0,0,0],[8.999999E+09,8.999999E+09,8.999999E+09,8.999999E+09,8.999999E+09,8.999999E+09]];
    CONST Robtarget Meulage_1_148 := [[-113.985,-31.1781,23],[0.636124910169873,-0.659503584363427,0.288259296349785,-0.278040822436365],[0,0,0,0],[8.999999E+09,8.999999E+09,8.999999E+09,8.999999E+09,8.999999E+09,8.999999E+09]];
    CONST Robtarget Meulage_1_149 := [[-110.183,-35.2679,23],[0.636265122297198,-0.659186926785766,0.288376691589601,-0.278349013741212],[0,0,0,0],[8.999999E+09,8.999999E+09,8.999999E+09,8.999999E+09,8.999999E+09,8.999999E+09]];
    CONST Robtarget Meulage_1_150 := [[-106.972,-38.7805,23],[0.6364508945365,-0.658915241369688,0.288387887231716,-0.278555901090681],[0,0,0,0],[8.999999E+09,8.999999E+09,8.999999E+09,8.999999E+09,8.999999E+09,8.999999E+09]];
    CONST Robtarget Meulage_1_151 := [[-103.269,-42.8101,23],[0.636680116491776,-0.658688881307593,0.28829567873108,-0.278662858183065],[0,0,0,0],[8.999999E+09,8.999999E+09,8.999999E+09,8.999999E+09,8.999999E+09,8.999999E+09]];
    CONST Robtarget Meulage_1_152 := [[-102.414,-43.7476,23],[0.636947415091093,-0.658497063362857,0.288117963776322,-0.278689158204359],[0,0,0,0],[8.999999E+09,8.999999E+09,8.999999E+09,8.999999E+09,8.999999E+09,8.999999E+09]];
    CONST Robtarget Meulage_1_153 := [[-93.6194,-53.2723,23],[0.637234505387833,-0.658330819071233,0.287888342023252,-0.278662915242101],[0,0,0,0],[8.999999E+09,8.999999E+09,8.999999E+09,8.999999E+09,8.999999E+09,8.999999E+09]];
    CONST Robtarget Meulage_1_154 := [[-92.358,-54.6464,23],[0.637529860811703,-0.658172281694406,0.287639810253692,-0.278618491381691],[0,0,0,0],[8.999999E+09,8.999999E+09,8.999999E+09,8.999999E+09,8.999999E+09,8.999999E+09]];
    CONST Robtarget Meulage_1_155 := [[-91.8745,-55.176,23],[0.63781449591397,-0.658010463475292,0.287408869737149,-0.278587581122084],[0,0,0,0],[8.999999E+09,8.999999E+09,8.999999E+09,8.999999E+09,8.999999E+09,8.999999E+09]];
    CONST Robtarget Meulage_1_156 := [[-89.8326,-57.5005,23],[0.638076265651583,-0.657834505246581,0.28722260580714,-0.278595796150037],[0,0,0,0],[8.999999E+09,8.999999E+09,8.999999E+09,8.999999E+09,8.999999E+09,8.999999E+09]];
    CONST Robtarget Meulage_1_157 := [[-78.5941,-69.5952,23],[0.638310478715851,-0.657633238677611,0.287098230423654,-0.278662631573636],[0,0,0,0],[8.999999E+09,8.999999E+09,8.999999E+09,8.999999E+09,8.999999E+09,8.999999E+09]];
    CONST Robtarget Meulage_1_158 := [[-77.0691,-71.2458,23],[0.638509169783228,-0.657406928951975,0.287046299030218,-0.278794892495759],[0,0,0,0],[8.999999E+09,8.999999E+09,8.999999E+09,8.999999E+09,8.999999E+09,8.999999E+09]];
    CONST Robtarget Meulage_1_159 := [[-73.6142,-75.1098,23],[0.638675271191981,-0.657155698201493,0.287062601325372,-0.278989872951453],[0,0,0,0],[8.999999E+09,8.999999E+09,8.999999E+09,8.999999E+09,8.999999E+09,8.999999E+09]];
    CONST Robtarget Meulage_1_160 := [[-71.0362,-77.9668,23],[0.638806902974317,-0.656892968215265,0.287136620676969,-0.27923096190772],[0,0,0,0],[8.999999E+09,8.999999E+09,8.999999E+09,8.999999E+09,8.999999E+09,8.999999E+09]];
    CONST Robtarget Meulage_1_161 := [[-69.5443,-79.5432,23],[0.638917079303558,-0.656626834458108,0.287242739785249,-0.279495571493358],[0,0,0,0],[8.999999E+09,8.999999E+09,8.999999E+09,8.999999E+09,8.999999E+09,8.999999E+09]];
    CONST Robtarget Meulage_1_162 := [[-62.4807,-87.1408,23],[0.639018831841439,-0.6563683370197,0.287352572926869,-0.279757104543038],[0,0,0,0],[8.999999E+09,8.999999E+09,8.999999E+09,8.999999E+09,8.999999E+09,8.999999E+09]];
    CONST Robtarget Meulage_1_163 := [[-62.0257,-87.6327,23],[0.639123652263771,-0.656135041356041,0.287433690881137,-0.279981495760296],[0,0,0,0],[8.999999E+09,8.999999E+09,8.999999E+09,8.999999E+09,8.999999E+09,8.999999E+09]];
    CONST Robtarget Meulage_1_164 := [[-61.4355,-88.2674,23],[0.639242016954097,-0.655936620973499,0.287462721158721,-0.280146349200464],[0,0,0,0],[8.999999E+09,8.999999E+09,8.999999E+09,8.999999E+09,8.999999E+09,8.999999E+09]];
    CONST Robtarget Meulage_1_165 := [[-57.1544,-92.8993,23],[0.639373999560924,-0.65578556878673,0.28742776232883,-0.280234647927723],[0,0,0,0],[8.999999E+09,8.999999E+09,8.999999E+09,8.999999E+09,8.999999E+09,8.999999E+09]];
    CONST Robtarget Meulage_1_166 := [[-56.2447,-93.9247,23],[0.639522074067197,-0.655678678482186,0.287328624510868,-0.280248548437522],[0,0,0,0],[8.999999E+09,8.999999E+09,8.999999E+09,8.999999E+09,8.999999E+09,8.999999E+09]];
    CONST Robtarget Meulage_1_167 := [[-50.657,-99.9769,23],[0.639676128681768,-0.655611125280001,0.287183701831911,-0.280203540673412],[0,0,0,0],[8.999999E+09,8.999999E+09,8.999999E+09,8.999999E+09,8.999999E+09,8.999999E+09]];
    CONST Robtarget Meulage_1_168 := [[-47.8722,-102.931,23],[0.639823179879182,-0.655568935057426,0.287024005180173,-0.280130131059292],[0,0,0,0],[8.999999E+09,8.999999E+09,8.999999E+09,8.999999E+09,8.999999E+09,8.999999E+09]];
    CONST Robtarget Meulage_1_169 := [[-44.884,-106.092,23],[0.639948554768623,-0.655539437549809,0.286881612690612,-0.280058624874266],[0,0,0,0],[8.999999E+09,8.999999E+09,8.999999E+09,8.999999E+09,8.999999E+09,8.999999E+09]];
    CONST Robtarget Meulage_1_170 := [[-43.8085,-107.276,23],[0.640038530889183,-0.655512653594342,0.286784767895676,-0.280014886850581],[0,0,0,0],[8.999999E+09,8.999999E+09,8.999999E+09,8.999999E+09,8.999999E+09,8.999999E+09]];
    CONST Robtarget Meulage_1_171 := [[-41.4395,-109.822,23],[0.640087073684898,-0.655482812147606,0.286747234981792,-0.280012221716958],[0,0,0,0],[8.999999E+09,8.999999E+09,8.999999E+09,8.999999E+09,8.999999E+09,8.999999E+09]];
    CONST Robtarget Meulage_1_172 := [[-36.95,-114.732,23],[0.640089043676979,-0.655453572453624,0.286772520139534,-0.280050267300876],[0,0,0,0],[8.999999E+09,8.999999E+09,8.999999E+09,8.999999E+09,8.999999E+09,8.999999E+09]];
    CONST Robtarget Meulage_1_173 := [[-34.1769,-117.743,23],[0.640051152525522,-0.655427286790841,0.286849224536431,-0.280119824831438],[0,0,0,0],[8.999999E+09,8.999999E+09,8.999999E+09,8.999999E+09,8.999999E+09,8.999999E+09]];
    CONST Robtarget Meulage_1_174 := [[-29.3842,-122.837,23],[0.639975547641572,-0.655412174735353,0.286966542928171,-0.280207749481342],[0,0,0,0],[8.999999E+09,8.999999E+09,8.999999E+09,8.999999E+09,8.999999E+09,8.999999E+09]];
    CONST Robtarget Meulage_1_175 := [[-26.5396,-125.852,23],[0.639867877066597,-0.655413417048551,0.287111816734701,-0.280301903922053],[0,0,0,0],[8.999999E+09,8.999999E+09,8.999999E+09,8.999999E+09,8.999999E+09,8.999999E+09]];
    CONST Robtarget Meulage_1_176 := [[-25.2028,-127.312,23],[0.63972639207889,-0.655437461018544,0.287281246609879,-0.280395013004092],[0,0,0,0],[8.999999E+09,8.999999E+09,8.999999E+09,8.999999E+09,8.999999E+09,8.999999E+09]];
    CONST Robtarget Meulage_1_177 := [[-23.2997,-129.413,23],[0.639550051682663,-0.65548590481334,0.287474698035776,-0.280485753600749],[0,0,0,0],[8.999999E+09,8.999999E+09,8.999999E+09,8.999999E+09,8.999999E+09,8.999999E+09]];
    CONST Robtarget Meulage_1_178 := [[-20.3176,-132.732,23],[0.639339337559082,-0.65555921659764,0.287691037178392,-0.280572971097758],[0,0,0,0],[8.999999E+09,8.999999E+09,8.999999E+09,8.999999E+09,8.999999E+09,8.999999E+09]];
    CONST Robtarget Meulage_1_179 := [[-19.9835,-133.099,23],[0.639094661632229,-0.655662116323942,0.287925162214809,-0.280649788267107],[0,0,0,0],[8.999999E+09,8.999999E+09,8.999999E+09,8.999999E+09,8.999999E+09,8.999999E+09]];
    CONST Robtarget Meulage_1_180 := [[-13.3873,-140.08,23],[0.638817676741106,-0.655805843252321,0.288164062628011,-0.280699385195136],[0,0,0,0],[8.999999E+09,8.999999E+09,8.999999E+09,8.999999E+09,8.999999E+09,8.999999E+09]];
    CONST Robtarget Meulage_1_181 := [[-8.98987,-144.815,23],[0.63851758051388,-0.656000678970394,0.288385388739874,-0.280699619035073],[0,0,0,0],[8.999999E+09,8.999999E+09,8.999999E+09,8.999999E+09,8.999999E+09,8.999999E+09]];
    CONST Robtarget Meulage_1_182 := [[-6.97433,-147.02,23],[0.638202411095335,-0.6562613904422,0.288564043002644,-0.280623347162955],[0,0,0,0],[8.999999E+09,8.999999E+09,8.999999E+09,8.999999E+09,8.999999E+09,8.999999E+09]];
    CONST Robtarget Meulage_1_183 := [[-5.94577,-148.175,23],[0.637879622513966,-0.656597143224025,0.288680957416832,-0.280451570714786],[0,0,0,0],[8.999999E+09,8.999999E+09,8.999999E+09,8.999999E+09,8.999999E+09,8.999999E+09]];
    CONST Robtarget Meulage_1_184 := [[-3.73541,-150.526,23],[0.637545024064339,-0.657019015227249,0.28873085314043,-0.280172893702116],[0,0,0,0],[8.999999E+09,8.999999E+09,8.999999E+09,8.999999E+09,8.999999E+09,8.999999E+09]];
    CONST Robtarget Meulage_1_185 := [[-1.71667,-152.753,23],[0.637197577946949,-0.657522981872248,0.28871844498612,-0.279793556918607],[0,0,0,0],[8.999999E+09,8.999999E+09,8.999999E+09,8.999999E+09,8.999999E+09,8.999999E+09]];
    CONST Robtarget Meulage_1_186 := [[0.872742,-155.514,23],[0.636823632161228,-0.658108506687163,0.28866210627579,-0.279326052038471],[0,0,0,0],[8.999999E+09,8.999999E+09,8.999999E+09,8.999999E+09,8.999999E+09,8.999999E+09]];
    CONST Robtarget Meulage_1_187 := [[4.61334,-159.486,23],[0.636410019324081,-0.65876698273121,0.288587292935696,-0.278793335865813],[0,0,0,0],[8.999999E+09,8.999999E+09,8.999999E+09,8.999999E+09,8.999999E+09,8.999999E+09]];
    CONST Robtarget Meulage_1_188 := [[7.81036,-162.948,23],[0.635940400807012,-0.659493510817619,0.288520256670746,-0.278216062263692],[0,0,0,0],[8.999999E+09,8.999999E+09,8.999999E+09,8.999999E+09,8.999999E+09,8.999999E+09]];
    CONST Robtarget Meulage_1_189 := [[12.5308,-168.197,23],[0.635401135129106,-0.660279391300196,0.288487378605509,-0.277617642245964],[0,0,0,0],[8.999999E+09,8.999999E+09,8.999999E+09,8.999999E+09,8.999999E+09,8.999999E+09]];
    CONST Robtarget Meulage_1_190 := [[13.6038,-169.382,23],[0.634775656761109,-0.661118590406087,0.288516566672985,-0.277020334557238],[0,0,0,0],[8.999999E+09,8.999999E+09,8.999999E+09,8.999999E+09,8.999999E+09,8.999999E+09]];
    CONST Robtarget Meulage_1_191 := [[15.4769,-171.371,23],[0.634048650828401,-0.662008366390557,0.288630894369783,-0.276440659142048],[0,0,0,0],[8.999999E+09,8.999999E+09,8.999999E+09,8.999999E+09,8.999999E+09,8.999999E+09]];
    CONST Robtarget Meulage_1_192 := [[19.7585,-175.906,23],[0.633208147143917,-0.662940531705686,0.288854306602718,-0.275899408062817],[0,0,0,0],[8.999999E+09,8.999999E+09,8.999999E+09,8.999999E+09,8.999999E+09,8.999999E+09]];
    CONST Robtarget Meulage_1_193 := [[20.0427,-176.209,23],[0.632242122571342,-0.663915084920475,0.289202744575249,-0.275405938555553],[0,0,0,0],[8.999999E+09,8.999999E+09,8.999999E+09,8.999999E+09,8.999999E+09,8.999999E+09]];
    CONST Robtarget Meulage_1_194 := [[20.4638,-176.658,23],[0.631139516633609,-0.664931874100008,0.289690877007776,-0.274968560253369],[0,0,0,0],[8.999999E+09,8.999999E+09,8.999999E+09,8.999999E+09,8.999999E+09,8.999999E+09]];
    CONST Robtarget Meulage_1_195 := [[20.5949,-176.806,23],[0.629894768237633,-0.665993308563411,0.290323150657496,-0.274586893510824],[0,0,0,0],[8.999999E+09,8.999999E+09,8.999999E+09,8.999999E+09,8.999999E+09,8.999999E+09]];
    CONST Robtarget Meulage_1_196 := [[29.2462,-186.139,23],[0.628506221975823,-0.667106650901289,0.291093585333216,-0.274250195695093],[0,0,0,0],[8.999999E+09,8.999999E+09,8.999999E+09,8.999999E+09,8.999999E+09,8.999999E+09]];
    CONST Robtarget Meulage_1_197 := [[30.8321,-187.832,23],[0.626974998709346,-0.668280617331141,0.291990675095576,-0.273943083778646],[0,0,0,0],[8.999999E+09,8.999999E+09,8.999999E+09,8.999999E+09,8.999999E+09,8.999999E+09]];
    CONST Robtarget Meulage_1_198 := [[34.5456,-191.818,23],[0.625305694697001,-0.669529245942158,0.292992506789379,-0.273639850849437],[0,0,0,0],[8.999999E+09,8.999999E+09,8.999999E+09,8.999999E+09,8.999999E+09,8.999999E+09]];
    CONST Robtarget Meulage_1_199 := [[37.9139,-195.429,23],[0.62350327865371,-0.670864380295598,0.294078571918561,-0.273317467969058],[0,0,0,0],[8.999999E+09,8.999999E+09,8.999999E+09,8.999999E+09,8.999999E+09,8.999999E+09]];
    CONST Robtarget Meulage_1_200 := [[41.6153,-199.46,23],[0.621571247499699,-0.672297765832567,0.295230151502326,-0.272954311162366],[0,0,0,0],[8.999999E+09,8.999999E+09,8.999999E+09,8.999999E+09,8.999999E+09,8.999999E+09]];
    CONST Robtarget Meulage_1_201 := [[45.3241,-203.521,23],[0.61950871145989,-0.673834774176657,0.296440676223087,-0.27254096759203],[0,0,0,0],[8.999999E+09,8.999999E+09,8.999999E+09,8.999999E+09,8.999999E+09,8.999999E+09]];
    CONST Robtarget Meulage_1_202 := [[48.2183,-206.733,23],[0.617311749592992,-0.675471768488509,0.297716698249405,-0.272082453261724],[0,0,0,0],[8.999999E+09,8.999999E+09,8.999999E+09,8.999999E+09,8.999999E+09,8.999999E+09]];
    CONST Robtarget Meulage_1_203 := [[54.3415,-213.565,23],[0.61497142430722,-0.677198933762205,0.299077810051921,-0.271595682829143],[0,0,0,0],[8.999999E+09,8.999999E+09,8.999999E+09,8.999999E+09,8.999999E+09,8.999999E+09]];
    CONST Robtarget Meulage_1_204 := [[56.373,-215.691,23],[0.612461700417115,-0.678993481697781,0.300580104030737,-0.271127494723371],[0,0,0,0],[8.999999E+09,8.999999E+09,8.999999E+09,8.999999E+09,8.999999E+09,8.999999E+09]];
    CONST Robtarget Meulage_1_205 := [[59.2057,-218.786,23],[0.609760124560934,-0.680827653502467,0.302280091144881,-0.270726879380679],[0,0,0,0],[8.999999E+09,8.999999E+09,8.999999E+09,8.999999E+09,8.999999E+09,8.999999E+09]];
    CONST Robtarget Meulage_1_206 := [[61.7748,-221.584,23],[0.606848060244874,-0.682673859887544,0.304228977058325,-0.270437723554464],[0,0,0,0],[8.999999E+09,8.999999E+09,8.999999E+09,8.999999E+09,8.999999E+09,8.999999E+09]];
    CONST Robtarget Meulage_1_207 := [[63.9059,-223.918,23],[0.603734691683607,-0.684531973125298,0.306411595457302,-0.270244951842206],[0,0,0,0],[8.999999E+09,8.999999E+09,8.999999E+09,8.999999E+09,8.999999E+09,8.999999E+09]];
    CONST Robtarget Meulage_1_208 := [[66.907,-227.265,23],[0.600445045984793,-0.686423190671066,0.308768872811463,-0.270093934111842],[0,0,0,0],[8.999999E+09,8.999999E+09,8.999999E+09,8.999999E+09,8.999999E+09,8.999999E+09]];
    CONST Robtarget Meulage_1_209 := [[68.9098,-229.444,23],[0.597071244277274,-0.688439054078672,0.311078050893575,-0.269792595022001],[0,0,0,0],[8.999999E+09,8.999999E+09,8.999999E+09,8.999999E+09,8.999999E+09,8.999999E+09]];
    CONST Robtarget Meulage_1_210 := [[71.5805,-232.309,23],[0.593756083971299,-0.69073198321376,0.312984249115269,-0.269042561537026],[0,0,0,0],[8.999999E+09,8.999999E+09,8.999999E+09,8.999999E+09,8.999999E+09,8.999999E+09]];
    CONST Robtarget Meulage_1_211 := [[73.5996,-234.524,23],[0.590716864018372,-0.693553209399158,0.31392286977493,-0.267376072468535],[0,0,0,0],[8.999999E+09,8.999999E+09,8.999999E+09,8.999999E+09,8.999999E+09,8.999999E+09]];
    CONST Robtarget Meulage_1_212 := [[77.5632,-238.995,23],[0.588226286650699,-0.697213713972814,0.313167645000666,-0.264213737088179],[0,0,0,0],[8.999999E+09,8.999999E+09,8.999999E+09,8.999999E+09,8.999999E+09,8.999999E+09]];
    CONST Robtarget Meulage_1_213 := [[77.5837,-239.019,23],[0.586583124034301,-0.702075014980479,0.309836057875843,-0.258867783198834],[0,0,0,0],[8.999999E+09,8.999999E+09,8.999999E+09,8.999999E+09,8.999999E+09,8.999999E+09]];
    CONST Robtarget Meulage_1_214 := [[77.6055,-239.043,23],[0.58607057560557,-0.708491768912966,0.302930583057703,-0.250586822559075],[0,0,0,0],[8.999999E+09,8.999999E+09,8.999999E+09,8.999999E+09,8.999999E+09,8.999999E+09]];
    CONST Robtarget Meulage_1_215 := [[77.619,-239.06,23],[0.586925901009966,-0.716782962438239,0.291289451652401,-0.23851756085862],[0,0,0,0],[8.999999E+09,8.999999E+09,8.999999E+09,8.999999E+09,8.999999E+09,8.999999E+09]];
    CONST Robtarget Meulage_1_216 := [[79.3052,-241.25,23],[0.58929101892533,-0.727148399615437,0.273567467193966,-0.221702821009869],[0,0,0,0],[8.999999E+09,8.999999E+09,8.999999E+09,8.999999E+09,8.999999E+09,8.999999E+09]];
    CONST Robtarget Meulage_1_217 := [[79.3694,-241.328,23],[0.593128711399467,-0.739581190004875,0.24819186251768,-0.199044704738873],[0,0,0,0],[8.999999E+09,8.999999E+09,8.999999E+09,8.999999E+09,8.999999E+09,8.999999E+09]];
    CONST Robtarget Meulage_1_218 := [[81.1309,-243.325,23],[0.598125560369574,-0.753725107253824,0.213294737748333,-0.169262020479093],[0,0,0,0],[8.999999E+09,8.999999E+09,8.999999E+09,8.999999E+09,8.999999E+09,8.999999E+09]];
    CONST Robtarget Meulage_1_219 := [[82.3723,-244.478,23],[0.60349456299872,-0.768593457201108,0.166953762216004,-0.131091003736161],[0,0,0,0],[8.999999E+09,8.999999E+09,8.999999E+09,8.999999E+09,8.999999E+09,8.999999E+09]];
    CONST Robtarget Meulage_1_220 := [[84.6533,-245.874,23],[0.607761916540144,-0.782283111303909,0.107868157829033,-0.083803622228985],[0,0,0,0],[8.999999E+09,8.999999E+09,8.999999E+09,8.999999E+09,8.999999E+09,8.999999E+09]];
    CONST Robtarget Meulage_1_221 := [[84.963,-246.064,23],[0.608804255507585,-0.791966130435412,0.0367360159937219,-0.0282398981571051],[0,0,0,0],[8.999999E+09,8.999999E+09,8.999999E+09,8.999999E+09,8.999999E+09,8.999999E+09]];
    CONST Robtarget Meulage_1_222 := [[87.6468,-245.799,23],[0.604582925870848,-0.794793010265326,-0.0419913029081179,0.0319419326106604],[0,0,0,0],[8.999999E+09,8.999999E+09,8.999999E+09,8.999999E+09,8.999999E+09,8.999999E+09]];
    CONST Robtarget Meulage_1_223 := [[88.2056,-245.724,23],[0.594550308059276,-0.789791257862159,-0.120475728560137,0.0906934342663952],[0,0,0,0],[8.999999E+09,8.999999E+09,8.999999E+09,8.999999E+09,8.999999E+09,8.999999E+09]];
    CONST Robtarget Meulage_1_224 := [[88.4192,-245.596,23],[0.580306489013225,-0.778830443855854,-0.190887558279981,0.142230301364883],[0,0,0,0],[8.999999E+09,8.999999E+09,8.999999E+09,8.999999E+09,8.999999E+09,8.999999E+09]];
    CONST Robtarget Meulage_1_225 := [[90.3592,-244.241,23],[0.56453883953836,-0.76536443320668,-0.248713188430869,0.183452808469782],[0,0,0,0],[8.999999E+09,8.999999E+09,8.999999E+09,8.999999E+09,8.999999E+09,8.999999E+09]];
    CONST Robtarget Meulage_1_226 := [[90.8914,-243.714,23],[0.549593092099443,-0.752502679303569,-0.293049940342331,0.21403009887135],[0,0,0,0],[8.999999E+09,8.999999E+09,8.999999E+09,8.999999E+09,8.999999E+09,8.999999E+09]];
    CONST Robtarget Meulage_1_227 := [[92.3948,-242.015,23],[0.536830879222293,-0.742159987374118,-0.325122805662872,0.235172960801558],[0,0,0,0],[8.999999E+09,8.999999E+09,8.999999E+09,8.999999E+09,8.999999E+09,8.999999E+09]];
    CONST Robtarget Meulage_1_228 := [[94.0028,-239.468,23],[0.526779344179813,-0.735129984891166,-0.346857169740468,0.248550863323853],[0,0,0,0],[8.999999E+09,8.999999E+09,8.999999E+09,8.999999E+09,8.999999E+09,8.999999E+09]];
    CONST Robtarget Meulage_1_229 := [[94.4142,-238.893,23],[0.519466744190544,-0.731545669288644,-0.360042872668452,0.255664556139004],[0,0,0,0],[8.999999E+09,8.999999E+09,8.999999E+09,8.999999E+09,8.999999E+09,8.999999E+09]];
    CONST Robtarget Meulage_1_230 := [[95.7895,-236.472,23],[0.514621527532025,-0.731102972294842,-0.366297433598701,0.257835834284644],[0,0,0,0],[8.999999E+09,8.999999E+09,8.999999E+09,8.999999E+09,8.999999E+09,8.999999E+09]];
    CONST Robtarget Meulage_1_231 := [[96.3749,-235.412,23],[0.511801380231035,-0.733247110466657,-0.367090966276298,0.256226939770664],[0,0,0,0],[8.999999E+09,8.999999E+09,8.999999E+09,8.999999E+09,8.999999E+09,8.999999E+09]];
    CONST Robtarget Meulage_1_232 := [[97.088,-234.415,23],[0.510517650498262,-0.737331991302475,-0.363720477816528,0.251834622616864],[0,0,0,0],[8.999999E+09,8.999999E+09,8.999999E+09,8.999999E+09,8.999999E+09,8.999999E+09]];
    CONST Robtarget Meulage_1_233 := [[98.3123,-232.682,23],[0.510252150195904,-0.742638424964313,-0.357490491714296,0.245624635004007],[0,0,0,0],[8.999999E+09,8.999999E+09,8.999999E+09,8.999999E+09,8.999999E+09,8.999999E+09]];
    CONST Robtarget Meulage_1_234 := [[100.573,-230.545,23],[0.510547227975904,-0.748514584831016,-0.349586654654341,0.238446252201535],[0,0,0,0],[8.999999E+09,8.999999E+09,8.999999E+09,8.999999E+09,8.999999E+09,8.999999E+09]];
    CONST Robtarget Meulage_1_235 := [[100.65,-230.467,23],[0.511054224117548,-0.75444591445731,-0.340997532035631,0.230988366191662],[0,0,0,0],[8.999999E+09,8.999999E+09,8.999999E+09,8.999999E+09,8.999999E+09,8.999999E+09]];
    CONST Robtarget Meulage_1_236 := [[100.679,-230.441,23],[0.511544924780465,-0.76008728112112,-0.33245603379348,0.223745615830924],[0,0,0,0],[8.999999E+09,8.999999E+09,8.999999E+09,8.999999E+09,8.999999E+09,8.999999E+09]];
    CONST Robtarget Meulage_1_237 := [[100.695,-230.428,23],[0.511901732137429,-0.765245812970092,-0.324431558597519,0.217024482841053],[0,0,0,0],[8.999999E+09,8.999999E+09,8.999999E+09,8.999999E+09,8.999999E+09,8.999999E+09]];
    CONST Robtarget Meulage_1_238 := [[100.74,-230.392,23],[0.512091790342682,-0.76986991257989,-0.317122765734446,0.210939487580668],[0,0,0,0],[8.999999E+09,8.999999E+09,8.999999E+09,8.999999E+09,8.999999E+09,8.999999E+09]];
    CONST Robtarget Meulage_1_239 := [[101.405,-229.813,23],[0.512133992245554,-0.773968154605517,-0.310577280812705,0.205508691509987],[0,0,0,0],[8.999999E+09,8.999999E+09,8.999999E+09,8.999999E+09,8.999999E+09,8.999999E+09]];
    CONST Robtarget Meulage_1_240 := [[107.989,-224.093,23],[0.512065407800635,-0.777585114372358,-0.304752526263205,0.200689575655268],[0,0,0,0],[8.999999E+09,8.999999E+09,8.999999E+09,8.999999E+09,8.999999E+09,8.999999E+09]];
    CONST Robtarget Meulage_1_241 := [[109.955,-222.414,23],[0.511930802174496,-0.780782437572254,-0.299551010965618,0.196404762654025],[0,0,0,0],[8.999999E+09,8.999999E+09,8.999999E+09,8.999999E+09,8.999999E+09,8.999999E+09]];
    CONST Robtarget Meulage_1_242 := [[111.763,-220.831,23],[0.511759745189493,-0.783607436510114,-0.294903517504826,0.192596116297586],[0,0,0,0],[8.999999E+09,8.999999E+09,8.999999E+09,8.999999E+09,8.999999E+09,8.999999E+09]];
    CONST Robtarget Meulage_1_243 := [[117.344,-216.053,23],[0.511582911671462,-0.786088761643208,-0.29075976816235,0.189225105422545],[0,0,0,0],[8.999999E+09,8.999999E+09,8.999999E+09,8.999999E+09,8.999999E+09,8.999999E+09]];
    CONST Robtarget Meulage_1_244 := [[120.652,-213.307,23],[0.511416800038009,-0.78825929599462,-0.287072824287811,0.186250724756627],[0,0,0,0],[8.999999E+09,8.999999E+09,8.999999E+09,8.999999E+09,8.999999E+09,8.999999E+09]];
    CONST Robtarget Meulage_1_245 := [[123.751,-210.756,23],[0.511279690302183,-0.790137998374649,-0.28381095701183,0.183647386284251],[0,0,0,0],[8.999999E+09,8.999999E+09,8.999999E+09,8.999999E+09,8.999999E+09,8.999999E+09]];
    CONST Robtarget Meulage_1_246 := [[125.281,-209.484,23],[0.511185392551123,-0.791749608461833,-0.280932246999438,0.181381158169022],[0,0,0,0],[8.999999E+09,8.999999E+09,8.999999E+09,8.999999E+09,8.999999E+09,8.999999E+09]];
    CONST Robtarget Meulage_1_247 := [[127.39,-207.786,23],[0.51114853586049,-0.793109626259566,-0.278405555632461,0.179428653272183],[0,0,0,0],[8.999999E+09,8.999999E+09,8.999999E+09,8.999999E+09,8.999999E+09,8.999999E+09]];
    CONST Robtarget Meulage_1_248 := [[129.386,-206.216,23],[0.511180387070529,-0.794240086521641,-0.276187828020938,0.177757082811338],[0,0,0,0],[8.999999E+09,8.999999E+09,8.999999E+09,8.999999E+09,8.999999E+09,8.999999E+09]];
    CONST Robtarget Meulage_1_249 := [[129.867,-205.834,23],[0.511290819530952,-0.795155183445355,-0.274249187162267,0.176344309361506],[0,0,0,0],[8.999999E+09,8.999999E+09,8.999999E+09,8.999999E+09,8.999999E+09,8.999999E+09]];
    CONST Robtarget Meulage_1_250 := [[134.318,-202.501,23],[0.511498833905872,-0.795872465294982,-0.272536600419235,0.175156396771989],[0,0,0,0],[8.999999E+09,8.999999E+09,8.999999E+09,8.999999E+09,8.999999E+09,8.999999E+09]];
    CONST Robtarget Meulage_1_251 := [[136.814,-200.653,23],[0.511817790011716,-0.796417285423537,-0.270986902838201,0.174149808487656],[0,0,0,0],[8.999999E+09,8.999999E+09,8.999999E+09,8.999999E+09,8.999999E+09,8.999999E+09]];
    CONST Robtarget Meulage_1_252 := [[137.667,-200.014,23],[0.512266087787594,-0.796816888256246,-0.269522794504857,0.17327367121037],[0,0,0,0],[8.999999E+09,8.999999E+09,8.999999E+09,8.999999E+09,8.999999E+09,8.999999E+09]];
    CONST Robtarget Meulage_1_253 := [[141.971,-196.782,23],[0.51287073114443,-0.79710000357277,-0.268048491811012,0.172467978122052],[0,0,0,0],[8.999999E+09,8.999999E+09,8.999999E+09,8.999999E+09,8.999999E+09,8.999999E+09]];
    CONST Robtarget Meulage_1_254 := [[144.391,-194.89,23],[0.513646710728389,-0.797290001920758,-0.266494627739153,0.171686699488559],[0,0,0,0],[8.999999E+09,8.999999E+09,8.999999E+09,8.999999E+09,8.999999E+09,8.999999E+09]];
    CONST Robtarget Meulage_1_255 := [[145.917,-193.75,23],[0.51461216663608,-0.797407346317784,-0.264791009163208,0.170884649558932],[0,0,0,0],[8.999999E+09,8.999999E+09,8.999999E+09,8.999999E+09,8.999999E+09,8.999999E+09]];
    CONST Robtarget Meulage_1_256 := [[147.858,-192.295,23],[0.515775395845837,-0.797466047566225,-0.262893620164732,0.17003113978285],[0,0,0,0],[8.999999E+09,8.999999E+09,8.999999E+09,8.999999E+09,8.999999E+09,8.999999E+09]];
    CONST Robtarget Meulage_1_257 := [[154.269,-187.738,23],[0.517158138387017,-0.797477665082862,-0.260741042943401,0.16908856294513],[0,0,0,0],[8.999999E+09,8.999999E+09,8.999999E+09,8.999999E+09,8.999999E+09,8.999999E+09]];
    CONST Robtarget Meulage_1_258 := [[155.109,-187.129,23],[0.518771821492135,-0.797467503376732,-0.258256855674741,0.168002305879447],[0,0,0,0],[8.999999E+09,8.999999E+09,8.999999E+09,8.999999E+09,8.999999E+09,8.999999E+09]];
    CONST Robtarget Meulage_1_259 := [[156.167,-186.367,23],[0.520654762328111,-0.797480825271707,-0.25527670118885,0.166663606162695],[0,0,0,0],[8.999999E+09,8.999999E+09,8.999999E+09,8.999999E+09,8.999999E+09,8.999999E+09]];
    CONST Robtarget Meulage_1_260 := [[161.3,-182.79,23],[0.522852260971845,-0.797575570527033,-0.251588862065417,0.164929581881895],[0,0,0,0],[8.999999E+09,8.999999E+09,8.999999E+09,8.999999E+09,8.999999E+09,8.999999E+09]];
    CONST Robtarget Meulage_1_261 := [[162.337,-182.044,23],[0.525435734954787,-0.797853865917615,-0.246827268753485,0.16255090425013],[0,0,0,0],[8.999999E+09,8.999999E+09,8.999999E+09,8.999999E+09,8.999999E+09,8.999999E+09]];
    CONST Robtarget Meulage_1_262 := [[166.265,-179.192,23],[0.528471297575051,-0.798405976975025,-0.240622322549176,0.15926983851608],[0,0,0,0],[8.999999E+09,8.999999E+09,8.999999E+09,8.999999E+09,8.999999E+09,8.999999E+09]];
    CONST Robtarget Meulage_1_263 := [[168.234,-177.856,23],[0.532000541936061,-0.799284141136274,-0.232672993010688,0.154866275964891],[0,0,0,0],[8.999999E+09,8.999999E+09,8.999999E+09,8.999999E+09,8.999999E+09,8.999999E+09]];
    CONST Robtarget Meulage_1_264 := [[171.416,-175.692,23],[0.536019681448152,-0.800462542709719,-0.222867489457882,0.149240413298995],[0,0,0,0],[8.999999E+09,8.999999E+09,8.999999E+09,8.999999E+09,8.999999E+09,8.999999E+09]];
    CONST Robtarget Meulage_1_265 := [[173.811,-174.023,23],[0.540449791018951,-0.801809871185841,-0.211434423266658,0.142514695784024],[0,0,0,0],[8.999999E+09,8.999999E+09,8.999999E+09,8.999999E+09,8.999999E+09,8.999999E+09]];
    CONST Robtarget Meulage_1_266 := [[176.931,-171.835,23],[0.545117751894382,-0.803076600336295,-0.199115884699906,0.135157223344101],[0,0,0,0],[8.999999E+09,8.999999E+09,8.999999E+09,8.999999E+09,8.999999E+09,8.999999E+09]];
    CONST Robtarget Meulage_1_267 := [[178.23,-171.072,23],[0.549827214467087,-0.803956218343679,-0.187035825579189,0.127914163280712],[0,0,0,0],[8.999999E+09,8.999999E+09,8.999999E+09,8.999999E+09,8.999999E+09,8.999999E+09]];
    CONST Robtarget Meulage_1_268 := [[179.73,-170.258,23],[0.554333557143317,-0.8041117172712,-0.176810284256886,0.12188837907281],[0,0,0,0],[8.999999E+09,8.999999E+09,8.999999E+09,8.999999E+09,8.999999E+09,8.999999E+09]];
    CONST Robtarget Meulage_1_269 := [[181.843,-169.477,23],[0.558422516913577,-0.803239807643307,-0.17020239763216,0.118326868720982],[0,0,0,0],[8.999999E+09,8.999999E+09,8.999999E+09,8.999999E+09,8.999999E+09,8.999999E+09]];
    CONST Robtarget Meulage_1_270 := [[181.899,-169.459,23],[0.561889320129514,-0.801087047534643,-0.168856499607087,0.118437395855626],[0,0,0,0],[8.999999E+09,8.999999E+09,8.999999E+09,8.999999E+09,8.999999E+09,8.999999E+09]];
    CONST Robtarget Meulage_1_271 := [[181.987,-169.439,23],[0.564513529788458,-0.797384612063464,-0.174099232933966,0.123254664098276],[0,0,0,0],[8.999999E+09,8.999999E+09,8.999999E+09,8.999999E+09,8.999999E+09,8.999999E+09]];
    CONST Robtarget Meulage_1_272 := [[186.123,-168.511,23],[0.565995726917746,-0.791770441012773,-0.186840612101165,0.133562687600066],[0,0,0,0],[8.999999E+09,8.999999E+09,8.999999E+09,8.999999E+09,8.999999E+09,8.999999E+09]];
    CONST Robtarget Meulage_1_273 := [[186.762,-168.378,23],[0.565909566638726,-0.783734778389299,-0.207501847004792,0.149830380829276],[0,0,0,0],[8.999999E+09,8.999999E+09,8.999999E+09,8.999999E+09,8.999999E+09,8.999999E+09]];
    CONST Robtarget Meulage_1_274 := [[187.599,-168.058,23],[0.563656645169882,-0.77253583241738,-0.236185429418457,0.17232532291407],[0,0,0,0],[8.999999E+09,8.999999E+09,8.999999E+09,8.999999E+09,8.999999E+09,8.999999E+09]];
    CONST Robtarget Meulage_1_275 := [[189.291,-167.373,23],[0.558412791275065,-0.757200195153599,-0.272715700963915,0.201119778857035],[0,0,0,0],[8.999999E+09,8.999999E+09,8.999999E+09,8.999999E+09,8.999999E+09,8.999999E+09]];
    CONST Robtarget Meulage_1_276 := [[190.89,-166.471,23],[0.549157956840237,-0.736520400189689,-0.316603142753397,0.236062891073859],[0,0,0,0],[8.999999E+09,8.999999E+09,8.999999E+09,8.999999E+09,8.999999E+09,8.999999E+09]];
    CONST Robtarget Meulage_1_277 := [[191.774,-165.9,23],[0.534687701464767,-0.709117856430176,-0.366996003618718,0.276721630744845],[0,0,0,0],[8.999999E+09,8.999999E+09,8.999999E+09,8.999999E+09,8.999999E+09,8.999999E+09]];
    CONST Robtarget Meulage_1_278 := [[192.169,-165.539,23],[0.513942946258028,-0.673872294504221,-0.422066775073148,0.321898145491065],[0,0,0,0],[8.999999E+09,8.999999E+09,8.999999E+09,8.999999E+09,8.999999E+09,8.999999E+09]];
    CONST Robtarget Meulage_1_279 := [[192.345,-165.303,23],[0.486771500243177,-0.630912903782295,-0.478333988859726,0.369051499784979],[0,0,0,0],[8.999999E+09,8.999999E+09,8.999999E+09,8.999999E+09,8.999999E+09,8.999999E+09]];
    CONST Robtarget Meulage_1_280 := [[194.263,-162.863,23],[0.454745682067368,-0.582567117485864,-0.531033069693872,0.414518753685282],[0,0,0,0],[8.999999E+09,8.999999E+09,8.999999E+09,8.999999E+09,8.999999E+09,8.999999E+09]];
    CONST Robtarget Meulage_1_281 := [[194.752,-159.626,23],[0.421210284805531,-0.533315360025361,-0.575693169210213,0.45468010475472],[0,0,0,0],[8.999999E+09,8.999999E+09,8.999999E+09,8.999999E+09,8.999999E+09,8.999999E+09]];
    CONST Robtarget Meulage_1_282 := [[194.765,-159.555,23],[0.389975925031052,-0.488006115316781,-0.610023938106001,0.487482927134116],[0,0,0,0],[8.999999E+09,8.999999E+09,8.999999E+09,8.999999E+09,8.999999E+09,8.999999E+09]];
    CONST Robtarget Meulage_1_283 := [[194.748,-159.489,23],[0.363716076879884,-0.44984979810702,-0.634297610028475,0.512847264274993],[0,0,0,0],[8.999999E+09,8.999999E+09,8.999999E+09,8.999999E+09,8.999999E+09,8.999999E+09]];
    CONST Robtarget Meulage_1_284 := [[193.463,-156.321,23],[0.34345120639483,-0.419873608221797,-0.650254084999702,0.531899470657704],[0,0,0,0],[8.999999E+09,8.999999E+09,8.999999E+09,8.999999E+09,8.999999E+09,8.999999E+09]];
    CONST Robtarget Meulage_1_285 := [[192.431,-154.867,23],[0.329028516928463,-0.397641914006589,-0.659900108759323,0.546033872330706],[0,0,0,0],[8.999999E+09,8.999999E+09,8.999999E+09,8.999999E+09,8.999999E+09,8.999999E+09]];
    CONST Robtarget Meulage_1_286 := [[191.775,-153.653,23],[0.319666276239996,-0.381974895275021,-0.664984543961394,0.556510743388615],[0,0,0,0],[8.999999E+09,8.999999E+09,8.999999E+09,8.999999E+09,8.999999E+09,8.999999E+09]];
    CONST Robtarget Meulage_1_287 := [[189.691,-150.726,23],[0.314343470604955,-0.37146049798951,-0.666879417609145,0.564337774112901],[0,0,0,0],[8.999999E+09,8.999999E+09,8.999999E+09,8.999999E+09,8.999999E+09,8.999999E+09]];
    CONST Robtarget Meulage_1_288 := [[189.465,-150.407,23],[0.312088487347658,-0.364808373671754,-0.666580764527338,0.570250568545241],[0,0,0,0],[8.999999E+09,8.999999E+09,8.999999E+09,8.999999E+09,8.999999E+09,8.999999E+09]];
    CONST Robtarget Meulage_1_289 := [[188.81,-149.44,23],[0.312007809788848,-0.360875936421254,-0.664840157156706,0.574810621487369],[0,0,0,0],[8.999999E+09,8.999999E+09,8.999999E+09,8.999999E+09,8.999999E+09,8.999999E+09]];
    CONST Robtarget Meulage_1_290 := [[187.806,-147.897,23],[0.313362990271011,-0.358740977222798,-0.662204544266969,0.578440739524646],[0,0,0,0],[8.999999E+09,8.999999E+09,8.999999E+09,8.999999E+09,8.999999E+09,8.999999E+09]];
    CONST Robtarget Meulage_1_291 := [[186.606,-145.945,23],[0.315623817557967,-0.357765490167812,-0.659045638811152,0.58141577704696],[0,0,0,0],[8.999999E+09,8.999999E+09,8.999999E+09,8.999999E+09,8.999999E+09,8.999999E+09]];
    CONST Robtarget Meulage_1_292 := [[183.451,-140.847,23],[0.318369246821468,-0.357453373406945,-0.655641853463804,0.583953652702742],[0,0,0,0],[8.999999E+09,8.999999E+09,8.999999E+09,8.999999E+09,8.999999E+09,8.999999E+09]];
    CONST Robtarget Meulage_1_293 := [[181.787,-138.135,23],[0.32132421810944,-0.357492103902482,-0.652172815486534,0.586191744435302],[0,0,0,0],[8.999999E+09,8.999999E+09,8.999999E+09,8.999999E+09,8.999999E+09,8.999999E+09]];
    CONST Robtarget Meulage_1_294 := [[181,-136.857,23],[0.324284891255122,-0.357656817306834,-0.64876907562051,0.588234304385683],[0,0,0,0],[8.999999E+09,8.999999E+09,8.999999E+09,8.999999E+09,8.999999E+09,8.999999E+09]];
    CONST Robtarget Meulage_1_295 := [[178.371,-132.672,23],[0.327122102529888,-0.357813340338817,-0.64551434853934,0.590145718735495],[0,0,0,0],[8.999999E+09,8.999999E+09,8.999999E+09,8.999999E+09,8.999999E+09,8.999999E+09]];
    CONST Robtarget Meulage_1_296 := [[176.726,-130.107,23],[0.329731858210899,-0.357855991984082,-0.642474417093109,0.591981937277436],[0,0,0,0],[8.999999E+09,8.999999E+09,8.999999E+09,8.999999E+09,8.999999E+09,8.999999E+09]];
    CONST Robtarget Meulage_1_297 := [[174.267,-125.988,23],[0.332069476275359,-0.357741932652709,-0.63967637410021,0.593771596631332],[0,0,0,0],[8.999999E+09,8.999999E+09,8.999999E+09,8.999999E+09,8.999999E+09,8.999999E+09]];
    CONST Robtarget Meulage_1_298 := [[173.286,-124.411,23],[0.334073627998889,-0.357415602023487,-0.637159131590713,0.595547764277909],[0,0,0,0],[8.999999E+09,8.999999E+09,8.999999E+09,8.999999E+09,8.999999E+09,8.999999E+09]];
    CONST Robtarget Meulage_1_299 := [[171.489,-121.389,23],[0.33572797630325,-0.35686786265694,-0.634932757525416,0.597321059356828],[0,0,0,0],[8.999999E+09,8.999999E+09,8.999999E+09,8.999999E+09,8.999999E+09,8.999999E+09]];
    CONST Robtarget Meulage_1_300 := [[170.785,-120.292,23],[0.337043101599051,-0.356112834332234,-0.632988391222542,0.599092057588692],[0,0,0,0],[8.999999E+09,8.999999E+09,8.999999E+09,8.999999E+09,8.999999E+09,8.999999E+09]];
    CONST Robtarget Meulage_1_301 := [[169.812,-118.638,23],[0.338052234789261,-0.355187838818752,-0.63130392383793,0.60084743609013],[0,0,0,0],[8.999999E+09,8.999999E+09,8.999999E+09,8.999999E+09,8.999999E+09,8.999999E+09]];
    CONST Robtarget Meulage_1_302 := [[167.934,-115.697,23],[0.338809585329961,-0.354151672928079,-0.62984572533376,0.602560386790878],[0,0,0,0],[8.999999E+09,8.999999E+09,8.999999E+09,8.999999E+09,8.999999E+09,8.999999E+09]];
    CONST Robtarget Meulage_1_303 := [[163.868,-109.135,23],[0.339390264396379,-0.353078977108922,-0.628566214771876,0.604196986093137],[0,0,0,0],[8.999999E+09,8.999999E+09,8.999999E+09,8.999999E+09,8.999999E+09,8.999999E+09]];
    CONST Robtarget Meulage_1_304 := [[162.071,-106.242,23],[0.339870929111039,-0.352047481000988,-0.627419613036908,0.605718541768927],[0,0,0,0],[8.999999E+09,8.999999E+09,8.999999E+09,8.999999E+09,8.999999E+09,8.999999E+09]];
    CONST Robtarget Meulage_1_305 := [[160.799,-104.245,23],[0.340323155050001,-0.35112228079871,-0.626360538750569,0.60709617817906],[0,0,0,0],[8.999999E+09,8.999999E+09,8.999999E+09,8.999999E+09,8.999999E+09,8.999999E+09]];
    CONST Robtarget Meulage_1_306 := [[158.153,-99.912,23],[0.340799409880622,-0.350353743696618,-0.625358593880477,0.608304730840241],[0,0,0,0],[8.999999E+09,8.999999E+09,8.999999E+09,8.999999E+09,8.999999E+09,8.999999E+09]];
    CONST Robtarget Meulage_1_307 := [[156.384,-97.0147,23],[0.341327973539136,-0.349759820656491,-0.624393373934935,0.609340788820308],[0,0,0,0],[8.999999E+09,8.999999E+09,8.999999E+09,8.999999E+09,8.999999E+09,8.999999E+09]];
    CONST Robtarget Meulage_1_308 := [[154.039,-93.3012,23],[0.341908155111453,-0.349333025865339,-0.623463357729664,0.610212005844282],[0,0,0,0],[8.999999E+09,8.999999E+09,8.999999E+09,8.999999E+09,8.999999E+09,8.999999E+09]];
    CONST Robtarget Meulage_1_309 := [[151.89,-89.8672,23],[0.342516156997653,-0.349040970864067,-0.622578927435569,0.610940718864773],[0,0,0,0],[8.999999E+09,8.999999E+09,8.999999E+09,8.999999E+09,8.999999E+09,8.999999E+09]];
    CONST Robtarget Meulage_1_310 := [[150.257,-87.1959,23],[0.343109642231483,-0.348832232843055,-0.62176027693475,0.611560303456279],[0,0,0,0],[8.999999E+09,8.999999E+09,8.999999E+09,8.999999E+09,8.999999E+09,8.999999E+09]];
    CONST Robtarget Meulage_1_311 := [[147.931,-83.3535,23],[0.343641888857798,-0.348652627127968,-0.621030464034866,0.612105187496111],[0,0,0,0],[8.999999E+09,8.999999E+09,8.999999E+09,8.999999E+09,8.999999E+09,8.999999E+09]];
    CONST Robtarget Meulage_1_312 := [[144.482,-77.5481,23],[0.344081191209919,-0.348459326635313,-0.620401234981102,0.612606349273618],[0,0,0,0],[8.999999E+09,8.999999E+09,8.999999E+09,8.999999E+09,8.999999E+09,8.999999E+09]];
    CONST Robtarget Meulage_1_313 := [[142.76,-74.793,23],[0.344411245302426,-0.348231887096648,-0.619879356924216,0.613078322710533],[0,0,0,0],[8.999999E+09,8.999999E+09,8.999999E+09,8.999999E+09,8.999999E+09,8.999999E+09]];
    CONST Robtarget Meulage_1_314 := [[140.805,-71.6352,23],[0.344645766954985,-0.347976287765885,-0.61945214567552,0.613523298409016],[0,0,0,0],[8.999999E+09,8.999999E+09,8.999999E+09,8.999999E+09,8.999999E+09,8.999999E+09]];
    CONST Robtarget Meulage_1_315 := [[138.523,-67.8589,23],[0.344818837513779,-0.34771943122809,-0.619095691472548,0.613931340820932],[0,0,0,0],[8.999999E+09,8.999999E+09,8.999999E+09,8.999999E+09,8.999999E+09,8.999999E+09]];
    CONST Robtarget Meulage_1_316 := [[136.963,-65.2217,23],[0.344972788052685,-0.347502442483784,-0.618785152511474,0.61428068747301],[0,0,0,0],[8.999999E+09,8.999999E+09,8.999999E+09,8.999999E+09,8.999999E+09,8.999999E+09]];
    CONST Robtarget Meulage_1_317 := [[136.39,-64.2772,23],[0.345155878874141,-0.347359492411539,-0.618484756152251,0.614561151324673],[0,0,0,0],[8.999999E+09,8.999999E+09,8.999999E+09,8.999999E+09,8.999999E+09,8.999999E+09]];
    CONST Robtarget Meulage_1_318 := [[135.1,-62.2359,23],[0.345391938890226,-0.347315152570696,-0.618181637540965,0.614758534996966],[0,0,0,0],[8.999999E+09,8.999999E+09,8.999999E+09,8.999999E+09,8.999999E+09,8.999999E+09]];
    CONST Robtarget Meulage_1_319 := [[128.658,-51.7282,23],[0.345683355983223,-0.347362426261735,-0.617868975900368,0.614882339019075],[0,0,0,0],[8.999999E+09,8.999999E+09,8.999999E+09,8.999999E+09,8.999999E+09,8.999999E+09]];
    CONST Robtarget Meulage_1_320 := [[126.874,-48.8117,23],[0.346002025876947,-0.347471472284848,-0.617561763647838,0.614950113519317],[0,0,0,0],[8.999999E+09,8.999999E+09,8.999999E+09,8.999999E+09,8.999999E+09,8.999999E+09]];
    CONST Robtarget Meulage_1_321 := [[122.779,-42.2419,23],[0.346305461388343,-0.347593555572849,-0.61728034743614,0.614992861914632],[0,0,0,0],[8.999999E+09,8.999999E+09,8.999999E+09,8.999999E+09,8.999999E+09,8.999999E+09]];
    CONST Robtarget Meulage_1_322 := [[122.753,-42.1998,23],[0.346546937628613,-0.347676091870017,-0.617047673633214,0.615043676193862],[0,0,0,0],[8.999999E+09,8.999999E+09,8.999999E+09,8.999999E+09,8.999999E+09,8.999999E+09]];
    CONST Robtarget Meulage_1_323 := [[122.731,-42.1644,23],[0.346691489985557,-0.347680568898709,-0.616881383436092,0.615126484189908],[0,0,0,0],[8.999999E+09,8.999999E+09,8.999999E+09,8.999999E+09,8.999999E+09,8.999999E+09]];
    CONST Robtarget Meulage_1_324 := [[120.79,-38.8672,23],[0.3467241348455,-0.347591479500586,-0.616789566610658,0.61525049225049],[0,0,0,0],[8.999999E+09,8.999999E+09,8.999999E+09,8.999999E+09,8.999999E+09,8.999999E+09]];
    CONST Robtarget Meulage_1_325 := [[116.939,-32.5593,23],[0.346657743406186,-0.347417723898329,-0.616762415761347,0.615413240483224],[0,0,0,0],[8.999999E+09,8.999999E+09,8.999999E+09,8.999999E+09,8.999999E+09,8.999999E+09]];
    CONST Robtarget Meulage_1_326 := [[115.219,-29.6957,23],[0.346520589304705,-0.347185731656406,-0.616782693475772,0.615601054215226],[0,0,0,0],[8.999999E+09,8.999999E+09,8.999999E+09,8.999999E+09,8.999999E+09,8.999999E+09]];
    CONST Robtarget Meulage_1_327 := [[114.481,-28.48,23],[0.346354529822173,-0.346933077927945,-0.616824074009089,0.615795453729511],[0,0,0,0],[8.999999E+09,8.999999E+09,8.999999E+09,8.999999E+09,8.999999E+09,8.999999E+09]];
    CONST Robtarget Meulage_1_328 := [[112.755,-25.5847,23],[0.346191270523437,-0.346693695005467,-0.61687000338882,0.615976042534044],[0,0,0,0],[8.999999E+09,8.999999E+09,8.999999E+09,8.999999E+09,8.999999E+09,8.999999E+09]];
    CONST Robtarget Meulage_1_329 := [[112.32,-24.8813,23],[0.346057319744365,-0.34648876539977,-0.616902358536721,0.616134195557201],[0,0,0,0],[8.999999E+09,8.999999E+09,8.999999E+09,8.999999E+09,8.999999E+09,8.999999E+09]];
    CONST Robtarget Meulage_1_330 := [[107.682,-17.3115,23],[0.345962799533024,-0.34632850923774,-0.616915572338982,0.616264133009624],[0,0,0,0],[8.999999E+09,8.999999E+09,8.999999E+09,8.999999E+09,8.999999E+09,8.999999E+09]];
    CONST Robtarget Meulage_1_331 := [[104.148,-11.4476,23],[0.345907168063966,-0.346211481501451,-0.616909469781888,0.616367217859588],[0,0,0,0],[8.999999E+09,8.999999E+09,8.999999E+09,8.999999E+09,8.999999E+09,8.999999E+09]];
    CONST Robtarget Meulage_1_332 := [[103.235,-9.93832,23],[0.345886984198449,-0.346134799243386,-0.616886378242296,0.616444718733113],[0,0,0,0],[8.999999E+09,8.999999E+09,8.999999E+09,8.999999E+09,8.999999E+09,8.999999E+09]];
    CONST Robtarget Meulage_1_333 := [[102.472,-8.69293,23],[0.345904649291364,-0.346098736157617,-0.61684368829224,0.616497771806796],[0,0,0,0],[8.999999E+09,8.999999E+09,8.999999E+09,8.999999E+09,8.999999E+09,8.999999E+09]];
    CONST Robtarget Meulage_1_334 := [[98.0627,-1.45071,23],[0.345965734925424,-0.34610895597016,-0.616778351662508,0.616523126715646],[0,0,0,0],[8.999999E+09,8.999999E+09,8.999999E+09,8.999999E+09,8.999999E+09,8.999999E+09]];
    CONST Robtarget Meulage_1_335 := [[94.6096,4.14087,23],[0.346076874798172,-0.346174492968982,-0.616688118834845,0.616514218194146],[0,0,0,0],[8.999999E+09,8.999999E+09,8.999999E+09,8.999999E+09,8.999999E+09,8.999999E+09]];
    CONST Robtarget Meulage_1_336 := [[92.8318,7.06226,23],[0.346247690467419,-0.346301488379856,-0.616565454874792,0.61646967147372],[0,0,0,0],[8.999999E+09,8.999999E+09,8.999999E+09,8.999999E+09,8.999999E+09,8.999999E+09]];
    CONST Robtarget Meulage_1_337 := [[89.2851,12.9241,23],[0.346472854723683,-0.346485277799896,-0.616413724594057,0.616391623352908],[0,0,0,0],[8.999999E+09,8.999999E+09,8.999999E+09,8.999999E+09,8.999999E+09,8.999999E+09]];
    CONST Robtarget Meulage_1_338 := [[84.41,20.8187,23],[0.346736659726748,-0.346711480035395,-0.616242516191281,0.616287270395423],[0,0,0,0],[8.999999E+09,8.999999E+09,8.999999E+09,8.999999E+09,8.999999E+09,8.999999E+09]];
    CONST Robtarget Meulage_1_339 := [[80.5696,26.9081,23],[0.347011448031713,-0.346954078942939,-0.616068339233552,0.616170206545078],[0,0,0,0],[8.999999E+09,8.999999E+09,8.999999E+09,8.999999E+09,8.999999E+09,8.999999E+09]];
    CONST Robtarget Meulage_1_340 := [[80.2197,27.466,23],[0.347262234952734,-0.347176271800177,-0.615909772858593,0.616062276212266],[0,0,0,0],[8.999999E+09,8.999999E+09,8.999999E+09,8.999999E+09,8.999999E+09,8.999999E+09]];
    CONST Robtarget Meulage_1_341 := [[80.0102,27.8116,23],[0.347454526423061,-0.347346331688659,-0.615787954875689,0.615979766356472],[0,0,0,0],[8.999999E+09,8.999999E+09,8.999999E+09,8.999999E+09,8.999999E+09,8.999999E+09]];
    CONST Robtarget Meulage_1_342 := [[78.2761,30.744,23],[0.347566402947449,-0.347440805418898,-0.615714359700723,0.615936936325764],[0,0,0,0],[8.999999E+09,8.999999E+09,8.999999E+09,8.999999E+09,8.999999E+09,8.999999E+09]];
    CONST Robtarget Meulage_1_343 := [[76.403,33.8336,23],[0.34759397435927,-0.347456876974281,-0.615691863401351,0.615934799287862],[0,0,0,0],[8.999999E+09,8.999999E+09,8.999999E+09,8.999999E+09,8.999999E+09,8.999999E+09]];
    CONST Robtarget Meulage_1_344 := [[73.8134,38.0974,23],[0.347550774667888,-0.347409860980394,-0.615713913689025,0.615963654780928],[0,0,0,0],[8.999999E+09,8.999999E+09,8.999999E+09,8.999999E+09,8.999999E+09,8.999999E+09]];
    CONST Robtarget Meulage_1_345 := [[71.1935,42.4257,23],[0.347463997037562,-0.34732779527077,-0.615765677955026,0.616007145451751],[0,0,0,0],[8.999999E+09,8.999999E+09,8.999999E+09,8.999999E+09,8.999999E+09,8.999999E+09]];
    CONST Robtarget Meulage_1_346 := [[69.6874,44.8746,23],[0.347366090852196,-0.347240545916251,-0.615827297855164,0.616049950421437],[0,0,0,0],[8.999999E+09,8.999999E+09,8.999999E+09,8.999999E+09,8.999999E+09,8.999999E+09]];
    CONST Robtarget Meulage_1_347 := [[67.7132,48.0794,23],[0.347278929302747,-0.347175902416773,-0.615890035872988,0.61607280556425],[0,0,0,0],[8.999999E+09,8.999999E+09,8.999999E+09,8.999999E+09,8.999999E+09,8.999999E+09]];
    CONST Robtarget Meulage_1_348 := [[66.7457,49.6413,23],[0.347214774594047,-0.347141487721623,-0.615944186598729,0.616074221828225],[0,0,0,0],[8.999999E+09,8.999999E+09,8.999999E+09,8.999999E+09,8.999999E+09,8.999999E+09]];
    CONST Robtarget Meulage_1_349 := [[65.8748,51.0194,23],[0.347167864915266,-0.347132948527447,-0.615993852280115,0.616055812057577],[0,0,0,0],[8.999999E+09,8.999999E+09,8.999999E+09,8.999999E+09,8.999999E+09,8.999999E+09]];
    CONST Robtarget Meulage_1_350 := [[61.9854,57.5121,23],[0.34711825840111,-0.347131137803491,-0.616050748491746,0.61602789152326],[0,0,0,0],[8.999999E+09,8.999999E+09,8.999999E+09,8.999999E+09,8.999999E+09,8.999999E+09]];
    CONST Robtarget Meulage_1_351 := [[60.3695,60.2164,23],[0.347041493871765,-0.347109904226762,-0.616127638469314,0.61600620859953],[0,0,0,0],[8.999999E+09,8.999999E+09,8.999999E+09,8.999999E+09,8.999999E+09,8.999999E+09]];
    CONST Robtarget Meulage_1_352 := [[57.9323,64.164,23],[0.346912082037728,-0.347050439769069,-0.616242943765075,0.615997267731034],[0,0,0,0],[8.999999E+09,8.999999E+09,8.999999E+09,8.999999E+09,8.999999E+09,8.999999E+09]];
    CONST Robtarget Meulage_1_353 := [[53.8799,70.843,23],[0.346720239149044,-0.346936712467966,-0.616398404427796,0.616013798810722],[0,0,0,0],[8.999999E+09,8.999999E+09,8.999999E+09,8.999999E+09,8.999999E+09,8.999999E+09]];
    CONST Robtarget Meulage_1_354 := [[51.6127,74.5532,23],[0.346461801946593,-0.346770400439421,-0.616599909343694,0.616051183724494],[0,0,0,0],[8.999999E+09,8.999999E+09,8.999999E+09,8.999999E+09,8.999999E+09,8.999999E+09]];
    CONST Robtarget Meulage_1_355 := [[48.9564,78.9262,23],[0.346146551940651,-0.346556874671432,-0.616839267720761,0.616108931111442],[0,0,0,0],[8.999999E+09,8.999999E+09,8.999999E+09,8.999999E+09,8.999999E+09,8.999999E+09]];
    CONST Robtarget Meulage_1_356 := [[46.438,83.0559,23],[0.345789536268692,-0.346313797322037,-0.617109587443843,0.616175386944629],[0,0,0,0],[8.999999E+09,8.999999E+09,8.999999E+09,8.999999E+09,8.999999E+09,8.999999E+09]];
    CONST Robtarget Meulage_1_357 := [[45.8388,84.0337,23],[0.345410752280685,-0.346061295522168,-0.617399698798159,0.616239080125849],[0,0,0,0],[8.999999E+09,8.999999E+09,8.999999E+09,8.999999E+09,8.999999E+09,8.999999E+09]];
    CONST Robtarget Meulage_1_358 := [[44.1538,86.751,23],[0.34503271866305,-0.34582116153544,-0.617696512262589,0.616288216685097],[0,0,0,0],[8.999999E+09,8.999999E+09,8.999999E+09,8.999999E+09,8.999999E+09,8.999999E+09]];
    CONST Robtarget Meulage_1_359 := [[40.9441,91.975,23],[0.344670886292617,-0.345617518419042,-0.617996671353378,0.616304003962549],[0,0,0,0],[8.999999E+09,8.999999E+09,8.999999E+09,8.999999E+09,8.999999E+09,8.999999E+09]];
    CONST Robtarget Meulage_1_360 := [[37.8567,96.9536,23],[0.344348490061225,-0.345463485429044,-0.618280965087153,0.616285441851963],[0,0,0,0],[8.999999E+09,8.999999E+09,8.999999E+09,8.999999E+09,8.999999E+09,8.999999E+09]];
    CONST Robtarget Meulage_1_361 := [[37.2034,98.0148,23],[0.344072948195446,-0.345374769075474,-0.618550297406678,0.616218796195205],[0,0,0,0],[8.999999E+09,8.999999E+09,8.999999E+09,8.999999E+09,8.999999E+09,8.999999E+09]];
    CONST Robtarget Meulage_1_362 := [[37.0622,98.2422,23],[0.343849474579666,-0.345356143226361,-0.618801437006315,0.616101821719447],[0,0,0,0],[8.999999E+09,8.999999E+09,8.999999E+09,8.999999E+09,8.999999E+09,8.999999E+09]];
    CONST Robtarget Meulage_1_363 := [[32.2876,106.065,23],[0.34367271037805,-0.345403155013592,-0.619037881581348,0.615936546906691],[0,0,0,0],[8.999999E+09,8.999999E+09,8.999999E+09,8.999999E+09,8.999999E+09,8.999999E+09]];
    CONST Robtarget Meulage_1_364 := [[30.3506,109.188,23],[0.343529856208066,-0.345504768250299,-0.619267820110154,0.615728073085831],[0,0,0,0],[8.999999E+09,8.999999E+09,8.999999E+09,8.999999E+09,8.999999E+09,8.999999E+09]];
    CONST Robtarget Meulage_1_365 := [[27.5604,113.703,23],[0.343398675669781,-0.345645794603767,-0.619507998579174,0.615480441539289],[0,0,0,0],[8.999999E+09,8.999999E+09,8.999999E+09,8.999999E+09,8.999999E+09,8.999999E+09]];
    CONST Robtarget Meulage_1_366 := [[26.9138,114.768,23],[0.343264944583604,-0.345803195997887,-0.61976100205868,0.615211856017814],[0,0,0,0],[8.999999E+09,8.999999E+09,8.999999E+09,8.999999E+09,8.999999E+09,8.999999E+09]];
    CONST Robtarget Meulage_1_367 := [[26.0292,116.245,23],[0.343108308038752,-0.345966430630852,-0.620044293708322,0.614921939494015],[0,0,0,0],[8.999999E+09,8.999999E+09,8.999999E+09,8.999999E+09,8.999999E+09,8.999999E+09]];
    CONST Robtarget Meulage_1_368 := [[25.6047,116.931,23],[0.342921983196896,-0.346132071665861,-0.620363745512009,0.614610385251436],[0,0,0,0],[8.999999E+09,8.999999E+09,8.999999E+09,8.999999E+09,8.999999E+09,8.999999E+09]];
    CONST Robtarget Meulage_1_369 := [[25.2603,117.502,23],[0.342706287306962,-0.346301847239865,-0.620720022535932,0.614275251708489],[0,0,0,0],[8.999999E+09,8.999999E+09,8.999999E+09,8.999999E+09,8.999999E+09,8.999999E+09]];
    CONST Robtarget Meulage_1_370 := [[23.8683,119.897,23],[0.342467598424788,-0.346482872061401,-0.621109912531141,0.613912078357153],[0,0,0,0],[8.999999E+09,8.999999E+09,8.999999E+09,8.999999E+09,8.999999E+09,8.999999E+09]];
    CONST Robtarget Meulage_1_371 := [[22.3846,122.287,23],[0.342210434628179,-0.346686179220246,-0.621534709130518,0.613510649390296],[0,0,0,0],[8.999999E+09,8.999999E+09,8.999999E+09,8.999999E+09,8.999999E+09,8.999999E+09]];
    CONST Robtarget Meulage_1_372 := [[19.572,126.883,23],[0.341940574705275,-0.346918804761765,-0.621991750788006,0.613066267400651],[0,0,0,0],[8.999999E+09,8.999999E+09,8.999999E+09,8.999999E+09,8.999999E+09,8.999999E+09]];
    CONST Robtarget Meulage_1_373 := [[18.1975,129.052,23],[0.34165686216022,-0.347186089355762,-0.622485449644773,0.61257185119562],[0,0,0,0],[8.999999E+09,8.999999E+09,8.999999E+09,8.999999E+09,8.999999E+09,8.999999E+09]];
    CONST Robtarget Meulage_1_374 := [[13.8513,136.071,23],[0.341360314029658,-0.347491852407717,-0.623016694842046,0.61202348522252],[0,0,0,0],[8.999999E+09,8.999999E+09,8.999999E+09,8.999999E+09,8.999999E+09,8.999999E+09]];
    CONST Robtarget Meulage_1_375 := [[11.9405,139.206,23],[0.341044338226029,-0.347840420427739,-0.623595559340875,0.611411792207973],[0,0,0,0],[8.999999E+09,8.999999E+09,8.999999E+09,8.999999E+09,8.999999E+09,8.999999E+09]];
    CONST Robtarget Meulage_1_376 := [[9.104,143.886,23],[0.340713761510459,-0.348233621829261,-0.624217144800109,0.610737614268737],[0,0,0,0],[8.999999E+09,8.999999E+09,8.999999E+09,8.999999E+09,8.999999E+09,8.999999E+09]];
    CONST Robtarget Meulage_1_377 := [[7.44629,146.522,23],[0.340371113238236,-0.348680243130038,-0.624883293904917,0.609992182181282],[0,0,0,0],[8.999999E+09,8.999999E+09,8.999999E+09,8.999999E+09,8.999999E+09,8.999999E+09]];
    CONST Robtarget Meulage_1_378 := [[4.77164,150.682,23],[0.34002190281736,-0.349190910987154,-0.625593277292224,0.609166532809542],[0,0,0,0],[8.999999E+09,8.999999E+09,8.999999E+09,8.999999E+09,8.999999E+09,8.999999E+09]];
    CONST Robtarget Meulage_1_379 := [[4.76913,150.686,23],[0.339667616246229,-0.349776799660013,-0.62635120777939,0.608248522732693],[0,0,0,0],[8.999999E+09,8.999999E+09,8.999999E+09,8.999999E+09,8.999999E+09,8.999999E+09]];
    CONST Robtarget Meulage_1_380 := [[-2.1944,162.086,23],[0.339307862412334,-0.350438784280475,-0.627157199707234,0.60723692232322],[0,0,0,0],[8.999999E+09,8.999999E+09,8.999999E+09,8.999999E+09,8.999999E+09,8.999999E+09]];
    CONST Robtarget Meulage_1_381 := [[-3.85391,164.784,23],[0.338932059435521,-0.351175368653461,-0.628021848685103,0.606126618052736],[0,0,0,0],[8.999999E+09,8.999999E+09,8.999999E+09,8.999999E+09,8.999999E+09,8.999999E+09]];
    CONST Robtarget Meulage_1_382 := [[-4.94791,166.582,23],[0.338531325585752,-0.35197729867299,-0.628949253894864,0.604922605662172],[0,0,0,0],[8.999999E+09,8.999999E+09,8.999999E+09,8.999999E+09,8.999999E+09,8.999999E+09]];
    CONST Robtarget Meulage_1_383 := [[-7.10254,170.098,23],[0.338090267845726,-0.352835399493637,-0.629951261209475,0.603625347506848],[0,0,0,0],[8.999999E+09,8.999999E+09,8.999999E+09,8.999999E+09,8.999999E+09,8.999999E+09]];
    CONST Robtarget Meulage_1_384 := [[-9.55142,174.134,23],[0.337602390948564,-0.353740316502347,-0.631029278154095,0.602241201030744],[0,0,0,0],[8.999999E+09,8.999999E+09,8.999999E+09,8.999999E+09,8.999999E+09,8.999999E+09]];
    CONST Robtarget Meulage_1_385 := [[-10.5059,175.739,23],[0.337060796046256,-0.354698452991093,-0.632194002747669,0.6007576633754],[0,0,0,0],[8.999999E+09,8.999999E+09,8.999999E+09,8.999999E+09,8.999999E+09,8.999999E+09]];
    CONST Robtarget Meulage_1_386 := [[-12.9516,179.667,23],[0.336469993699686,-0.355710220067256,-0.63343929099487,0.599176808048638],[0,0,0,0],[8.999999E+09,8.999999E+09,8.999999E+09,8.999999E+09,8.999999E+09,8.999999E+09]];
    CONST Robtarget Meulage_1_387 := [[-14.6994,182.494,23],[0.335834831694758,-0.356784418644583,-0.634763053658173,0.597491179971346],[0,0,0,0],[8.999999E+09,8.999999E+09,8.999999E+09,8.999999E+09,8.999999E+09,8.999999E+09]];
    CONST Robtarget Meulage_1_388 := [[-16.0259,184.679,23],[0.335140360293567,-0.357905973899579,-0.636173344592719,0.595707754170621],[0,0,0,0],[8.999999E+09,8.999999E+09,8.999999E+09,8.999999E+09,8.999999E+09,8.999999E+09]];
    CONST Robtarget Meulage_1_389 := [[-21.3898,193.343,23],[0.334376454832155,-0.359064346044699,-0.637675265228075,0.593831152744345],[0,0,0,0],[8.999999E+09,8.999999E+09,8.999999E+09,8.999999E+09,8.999999E+09,8.999999E+09]];
    CONST Robtarget Meulage_1_390 := [[-22.1974,194.651,23],[0.333498200978262,-0.360203182546081,-0.639291065250484,0.591894881815039],[0,0,0,0],[8.999999E+09,8.999999E+09,8.999999E+09,8.999999E+09,8.999999E+09,8.999999E+09]];
    CONST Robtarget Meulage_1_391 := [[-27.4388,203.37,23],[0.332440104351115,-0.361253439883216,-0.641062034023409,0.589931350010603],[0,0,0,0],[8.999999E+09,8.999999E+09,8.999999E+09,8.999999E+09,8.999999E+09,8.999999E+09]];
    CONST Robtarget Meulage_1_392 := [[-29.8692,207.379,23],[0.331106764447849,-0.362101192211458,-0.643043628141271,0.588001640680388],[0,0,0,0],[8.999999E+09,8.999999E+09,8.999999E+09,8.999999E+09,8.999999E+09,8.999999E+09]];
    CONST Robtarget Meulage_1_393 := [[-30.7266,208.84,23],[0.329398444912859,-0.362631917232335,-0.64529895192664,0.586160404442138],[0,0,0,0],[8.999999E+09,8.999999E+09,8.999999E+09,8.999999E+09,8.999999E+09,8.999999E+09]];
    CONST Robtarget Meulage_1_394 := [[-33.2451,213.202,23],[0.327132958677688,-0.362613174635372,-0.647931680894581,0.58453421612491],[0,0,0,0],[8.999999E+09,8.999999E+09,8.999999E+09,8.999999E+09,8.999999E+09,8.999999E+09]];
    CONST Robtarget Meulage_1_395 := [[-34.1776,214.73,23],[0.324129087029825,-0.361836185915462,-0.651059426339653,0.583212253710127],[0,0,0,0],[8.999999E+09,8.999999E+09,8.999999E+09,8.999999E+09,8.999999E+09,8.999999E+09]];
    CONST Robtarget Meulage_1_396 := [[-35.2131,216.436,23],[0.320091787531094,-0.359934300761062,-0.654856126799257,0.582367581415956],[0,0,0,0],[8.999999E+09,8.999999E+09,8.999999E+09,8.999999E+09,8.999999E+09,8.999999E+09]];
    CONST Robtarget Meulage_1_397 := [[-36.7297,218.828,23],[0.314675013357187,-0.35647594541557,-0.659520047239482,0.58218368544469],[0,0,0,0],[8.999999E+09,8.999999E+09,8.999999E+09,8.999999E+09,8.999999E+09,8.999999E+09]];
    CONST Robtarget Meulage_1_398 := [[-37.1261,219.435,23],[0.307484488650724,-0.350964369534354,-0.665260193076112,0.582843183081771],[0,0,0,0],[8.999999E+09,8.999999E+09,8.999999E+09,8.999999E+09,8.999999E+09,8.999999E+09]];
    CONST Robtarget Meulage_1_399 := [[-37.4698,219.976,23],[0.298139848743018,-0.342900081678875,-0.672238921291226,0.584488663087078],[0,0,0,0],[8.999999E+09,8.999999E+09,8.999999E+09,8.999999E+09,8.999999E+09,8.999999E+09]];
    CONST Robtarget Meulage_1_400 := [[-41.2437,226.036,23],[0.286273867123043,-0.331781035656909,-0.680554171401625,0.587209193702462],[0,0,0,0],[8.999999E+09,8.999999E+09,8.999999E+09,8.999999E+09,8.999999E+09,8.999999E+09]];
    CONST Robtarget Meulage_1_401 := [[-42.7228,228.797,23],[0.271652571225599,-0.317243554357959,-0.690154321798014,0.590972435794067],[0,0,0,0],[8.999999E+09,8.999999E+09,8.999999E+09,8.999999E+09,8.999999E+09,8.999999E+09]];
    CONST Robtarget Meulage_1_402 := [[-43.5453,230.427,23],[0.254000896825062,-0.298886436582636,-0.700941662633163,0.595677117257374],[0,0,0,0],[8.999999E+09,8.999999E+09,8.999999E+09,8.999999E+09,8.999999E+09,8.999999E+09]];
    CONST Robtarget Meulage_1_403 := [[-44.4672,232.089,23],[0.233012314462308,-0.27624235301284,-0.712721306898335,0.601185297894067],[0,0,0,0],[8.999999E+09,8.999999E+09,8.999999E+09,8.999999E+09,8.999999E+09,8.999999E+09]];
    CONST Robtarget Meulage_1_404 := [[-44.8771,232.71,23],[0.208320148439245,-0.248776983345834,-0.72521047620316,0.607274644223504],[0,0,0,0],[8.999999E+09,8.999999E+09,8.999999E+09,8.999999E+09,8.999999E+09,8.999999E+09]];
    CONST Robtarget Meulage_1_405 := [[-45.723,234.231,23],[0.1793419021249,-0.215693927006582,-0.738055228088528,0.61366692291983],[0,0,0,0],[8.999999E+09,8.999999E+09,8.999999E+09,8.999999E+09,8.999999E+09,8.999999E+09]];
    CONST Robtarget Meulage_1_406 := [[-45.7795,234.302,23],[0.145553944870429,-0.176256293237217,-0.750651912397005,0.619894728677097],[0,0,0,0],[8.999999E+09,8.999999E+09,8.999999E+09,8.999999E+09,8.999999E+09,8.999999E+09]];
    CONST Robtarget Meulage_1_407 := [[-46.5135,235.334,23],[0.106955042313489,-0.130359436652087,-0.762022499725197,0.625210961285895],[0,0,0,0],[8.999999E+09,8.999999E+09,8.999999E+09,8.999999E+09,8.999999E+09,8.999999E+09]];
    CONST Robtarget Meulage_1_408 := [[-47.8592,236.36,23],[0.0645853227056262,-0.0792023444693337,-0.770937214186033,0.628658521380766],[0,0,0,0],[8.999999E+09,8.999999E+09,8.999999E+09,8.999999E+09,8.999999E+09,8.999999E+09]];
    CONST Robtarget Meulage_1_409 := [[-49.3042,237.037,23],[0.0209725143572198,-0.025866423427946,-0.776328787855864,0.629447928685787],[0,0,0,0],[8.999999E+09,8.999999E+09,8.999999E+09,8.999999E+09,8.999999E+09,8.999999E+09]];
    CONST Robtarget Meulage_1_410 := [[-49.7381,237.127,23],[0.0203903987508376,-0.0252808280908948,0.777962749733697,-0.627470374915506],[0,0,0,0],[8.999999E+09,8.999999E+09,8.999999E+09,8.999999E+09,8.999999E+09,8.999999E+09]];
    CONST Robtarget Meulage_1_411 := [[-50.9257,237.05,23],[0.0564414116026378,-0.0703102848882154,0.776646408051886,-0.623451030759709],[0,0,0,0],[8.999999E+09,8.999999E+09,8.999999E+09,8.999999E+09,8.999999E+09,8.999999E+09]];
    CONST Robtarget Meulage_1_412 := [[-52.0769,236.8,23],[0.085623720724947,-0.107111644449848,0.773723191110182,-0.61850472723395],[0,0,0,0],[8.999999E+09,8.999999E+09,8.999999E+09,8.999999E+09,8.999999E+09,8.999999E+09]];
    CONST Robtarget Meulage_1_413 := [[-52.5359,236.567,23],[0.107759905929224,-0.135291468751757,0.770412779952729,-0.613635208933308],[0,0,0,0],[8.999999E+09,8.999999E+09,8.999999E+09,8.999999E+09,8.999999E+09,8.999999E+09]];
    CONST Robtarget Meulage_1_414 := [[-53.7056,235.903,23],[0.123691996835932,-0.155760625151689,0.767464814001796,-0.609456049966102],[0,0,0,0],[8.999999E+09,8.999999E+09,8.999999E+09,8.999999E+09,8.999999E+09,8.999999E+09]];
    CONST Robtarget Meulage_1_415 := [[-55.425,234.672,23],[0.134579773998135,-0.16987167319351,0.765196866350101,-0.606222446635749],[0,0,0,0],[8.999999E+09,8.999999E+09,8.999999E+09,8.999999E+09,8.999999E+09,8.999999E+09]];
    CONST Robtarget Meulage_1_416 := [[-56.5923,233.913,23],[0.141492630207116,-0.178902842855392,0.763666100425554,-0.603976568648287],[0,0,0,0],[8.999999E+09,8.999999E+09,8.999999E+09,8.999999E+09,8.999999E+09,8.999999E+09]];
    CONST Robtarget Meulage_1_417 := [[-57.8191,233.131,23],[0.145279147854607,-0.183876296663979,0.762797596874819,-0.602680099991513],[0,0,0,0],[8.999999E+09,8.999999E+09,8.999999E+09,8.999999E+09,8.999999E+09,8.999999E+09]];
    CONST Robtarget Meulage_1_418 := [[-58.3575,232.789,23],[0.146510408580604,-0.1854981842042,0.762511070385371,-0.602247450284553],[0,0,0,0],[8.999999E+09,8.999999E+09,8.999999E+09,8.999999E+09,8.999999E+09,8.999999E+09]];
    CONST Robtarget Meulage_1_419 := [[-58.3575,232.789,23],[0.148181865705,-0.238974835253123,0.815584650429269,-0.505722098366382],[0,0,0,0],[8.999999E+09,8.999999E+09,8.999999E+09,8.999999E+09,8.999999E+09,8.999999E+09]];
    !
    !Declaration des points de tronconnage

    !Tronconnage_1 : Tronconnage
    CONST Robtarget Tronconnage_0 := [[92.3768,-182.114,42.014],[0.999961923064171,0,0,0.00872653549837393],[0,0,0,0],[8.999999E+09,8.999999E+09,8.999999E+09,8.999999E+09,8.999999E+09,8.999999E+09]];

    !
    !Cycle
    PROC Cycle()
        !
        Prise;
        !
        Tronconnage;
        !
        Meulage;
        !
        !
        Depose;
        !
    ENDPROC

    !Trajectoire de prise de la pièce
    PROC PRISE()

		!
        !Trigger localisation
        LocalisationPieceTable 6 \model:=5;
        !
        !Approche
		MoveJ Reltool(PicKPosition,0,0,-200),V1000,Z0,Tool_Prehenseur \Wobj:=Wobj_vision;
		MoveL Reltool(PicKPosition,0,0,-100),V500,Z0,Tool_Prehenseur \Wobj:=Wobj_vision;
		MoveL Reltool(PicKPosition,0,0,-10),V200,Z0,Tool_Prehenseur \Wobj:=Wobj_vision;
		MoveL PicKPosition,V100,Fine,Tool_Prehenseur \Wobj:=Wobj_vision;

        !Fermeture pince
		Gripper_Close;
        !
		MoveL Reltool(PicKPosition,0,0,-200),V500,Z0,Tool_Prehenseur \Wobj:=Wobj_vision;

        !Trigger relocalisation
		LocalisationPiecePrehenseur 6 \model:=5,Ref;
        !
        PEO;
        !
    ENDPROC

    !Trajectoire de tronconnage
    PROC Tronconnage()
        !
        !StartMotor1();
        !
        !Trajectoire
            !---------- tronconnage zone : 1 ------------
            !Approche
            MoveJ Reltool(Tronconnage_0,-200,0,-300),V1000,Z0,Tool_M2_D490_S180 \Wobj:=Wobj_Part_0;
            MoveL Reltool(Tronconnage_0,0,0,-300),V500,Z0,Tool_M2_D490_S180 \Wobj:=Wobj_Part_0;
            MoveL Reltool(Tronconnage_0,0,0,-200),V500,Z0,Tool_M2_D490_S180 \Wobj:=Wobj_Part_0;
            MoveL Reltool(Tronconnage_0,0,0,-150),V100,Z0,Tool_M2_D490_S180 \Wobj:=Wobj_Part_0;
            !
            Movel reltool(Tronconnage_0,0,0,-28.4161),V100,Z0,Tool_M2_D490_S180 \Wobj:=Wobj_Part_0;
            Movel Tronconnage_0,V100,Z0,Tool_M2_D490_S180 \Wobj:=Wobj_Part_0;
            Movel reltool(Tronconnage_0,0,0,28.4161),V100,Z0,Tool_M2_D490_S180 \Wobj:=Wobj_Part_0;
            !
            !Degagement
            MoveL Reltool(Tronconnage_0,0,0,-150),V100,Z0,Tool_M2_D490_S180 \Wobj:=Wobj_Part_0;
            MoveL Reltool(Tronconnage_0,0,0,-200),V500,Z0,Tool_M2_D490_S180 \Wobj:=Wobj_Part_0;
            MoveL Reltool(Tronconnage_0,0,0,-300),V500,Z0,Tool_M2_D490_S180 \Wobj:=Wobj_Part_0;
            MoveJ Reltool(Tronconnage_0,-200,0,-300),V1000,Z0,Tool_M2_D490_S180 \Wobj:=Wobj_Part_0;
            !

    ENDPROC


    !Trajectoire de meulage
    PROC Meulage()
        !
        !StartMotor2();
        !

